  PROC DrawPart34()
    MoveL Offs(pOrigin,325.18,181.23,0.00),v40,z0,tPen\WObj:=wPaper;
    MoveL Offs(pOrigin,324.70,181.70,0.00),v40,z0,tPen\WObj:=wPaper;
    MoveL Offs(pOrigin,325.66,180.75,0.00),v40,z0,tPen\WObj:=wPaper;
    MoveL Offs(pOrigin,325.66,181.23,0.00),v40,z0,tPen\WObj:=wPaper;
    MoveL Offs(pOrigin,325.18,181.23,0.00),v40,z0,tPen\WObj:=wPaper;
    MoveL Offs(pOrigin,324.70,181.70,0.00),v40,fine,tPen\WObj:=wPaper;
    MoveL Offs(pOrigin,324.70,181.70,6.00),v60,z5,tPen\WObj:=wPaper;
    MoveL Offs(pOrigin,326.14,180.27,6.00),vTravel,z5,tPen\WObj:=wPaper;
    MoveL Offs(pOrigin,326.14,180.27,0.00),v60,z0,tPen\WObj:=wPaper;
    MoveL Offs(pOrigin,327.10,179.31,0.00),v40,z0,tPen\WObj:=wPaper;
    MoveL Offs(pOrigin,327.10,179.79,0.00),v40,z0,tPen\WObj:=wPaper;
    MoveL Offs(pOrigin,326.62,179.79,0.00),v40,z0,tPen\WObj:=wPaper;
    MoveL Offs(pOrigin,326.14,180.27,0.00),v40,z0,tPen\WObj:=wPaper;
    MoveL Offs(pOrigin,327.10,179.31,0.00),v40,z0,tPen\WObj:=wPaper;
    MoveL Offs(pOrigin,327.10,179.79,0.00),v40,z0,tPen\WObj:=wPaper;
    MoveL Offs(pOrigin,326.62,179.79,0.00),v40,z0,tPen\WObj:=wPaper;
    MoveL Offs(pOrigin,326.14,180.27,0.00),v40,fine,tPen\WObj:=wPaper;
    MoveL Offs(pOrigin,326.14,180.27,6.00),v60,z5,tPen\WObj:=wPaper;
    MoveL Offs(pOrigin,287.35,170.21,6.00),vTravel,z5,tPen\WObj:=wPaper;
    MoveL Offs(pOrigin,287.35,170.21,0.00),v60,z0,tPen\WObj:=wPaper;
    MoveL Offs(pOrigin,288.31,171.17,0.00),v40,z0,tPen\WObj:=wPaper;
    MoveL Offs(pOrigin,287.35,170.21,0.00),v40,fine,tPen\WObj:=wPaper;
    MoveL Offs(pOrigin,287.35,170.21,6.00),v60,z5,tPen\WObj:=wPaper;
    MoveL Offs(pOrigin,283.52,160.63,6.00),vTravel,z5,tPen\WObj:=wPaper;
    MoveL Offs(pOrigin,283.52,160.63,0.00),v60,z0,tPen\WObj:=wPaper;
    MoveL Offs(pOrigin,283.04,159.68,0.00),v40,z0,tPen\WObj:=wPaper;
    MoveL Offs(pOrigin,283.52,160.15,0.00),v40,z0,tPen\WObj:=wPaper;
    MoveL Offs(pOrigin,283.52,160.63,0.00),v40,z0,tPen\WObj:=wPaper;
    MoveL Offs(pOrigin,283.04,159.68,0.00),v40,z0,tPen\WObj:=wPaper;
    MoveL Offs(pOrigin,283.52,160.15,0.00),v40,z0,tPen\WObj:=wPaper;
    MoveL Offs(pOrigin,283.52,160.63,0.00),v40,fine,tPen\WObj:=wPaper;
    MoveL Offs(pOrigin,283.52,160.63,6.00),v60,z5,tPen\WObj:=wPaper;
    MoveL Offs(pOrigin,282.56,158.72,6.00),vTravel,z5,tPen\WObj:=wPaper;
    MoveL Offs(pOrigin,282.56,158.72,0.00),v60,z0,tPen\WObj:=wPaper;
    MoveL Offs(pOrigin,282.08,157.76,0.00),v40,z0,tPen\WObj:=wPaper;
    MoveL Offs(pOrigin,282.56,158.24,0.00),v40,z0,tPen\WObj:=wPaper;
    MoveL Offs(pOrigin,282.56,158.72,0.00),v40,z0,tPen\WObj:=wPaper;
    MoveL Offs(pOrigin,282.08,157.76,0.00),v40,z0,tPen\WObj:=wPaper;
    MoveL Offs(pOrigin,282.56,158.24,0.00),v40,z0,tPen\WObj:=wPaper;
    MoveL Offs(pOrigin,282.56,158.72,0.00),v40,fine,tPen\WObj:=wPaper;
    MoveL Offs(pOrigin,282.56,158.72,6.00),v60,z5,tPen\WObj:=wPaper;
    MoveL Offs(pOrigin,276.82,149.62,6.00),vTravel,z5,tPen\WObj:=wPaper;
    MoveL Offs(pOrigin,276.82,149.62,0.00),v60,z0,tPen\WObj:=wPaper;
    MoveL Offs(pOrigin,277.77,150.58,0.00),v40,z0,tPen\WObj:=wPaper;
    MoveL Offs(pOrigin,276.82,149.62,0.00),v40,fine,tPen\WObj:=wPaper;
    MoveL Offs(pOrigin,276.82,149.62,6.00),v60,z5,tPen\WObj:=wPaper;
    MoveL Offs(pOrigin,275.38,147.70,6.00),vTravel,z5,tPen\WObj:=wPaper;
    MoveL Offs(pOrigin,275.38,147.70,0.00),v60,z0,tPen\WObj:=wPaper;
    MoveL Offs(pOrigin,276.34,148.66,0.00),v40,z0,tPen\WObj:=wPaper;
    MoveL Offs(pOrigin,275.38,147.70,0.00),v40,fine,tPen\WObj:=wPaper;
    MoveL Offs(pOrigin,275.38,147.70,6.00),v60,z5,tPen\WObj:=wPaper;
    MoveL Offs(pOrigin,300.28,147.23,6.00),vTravel,z5,tPen\WObj:=wPaper;
    MoveL Offs(pOrigin,300.28,147.23,0.00),v60,z0,tPen\WObj:=wPaper;
    MoveL Offs(pOrigin,300.76,146.27,0.00),v40,z0,tPen\WObj:=wPaper;
    MoveL Offs(pOrigin,300.76,146.75,0.00),v40,z0,tPen\WObj:=wPaper;
    MoveL Offs(pOrigin,300.28,147.23,0.00),v40,z0,tPen\WObj:=wPaper;
    MoveL Offs(pOrigin,300.76,146.27,0.00),v40,z0,tPen\WObj:=wPaper;
    MoveL Offs(pOrigin,300.76,146.75,0.00),v40,z0,tPen\WObj:=wPaper;
    MoveL Offs(pOrigin,300.28,147.23,0.00),v40,fine,tPen\WObj:=wPaper;
    MoveL Offs(pOrigin,300.28,147.23,6.00),v60,z5,tPen\WObj:=wPaper;
    MoveL Offs(pOrigin,301.24,145.79,6.00),vTravel,z5,tPen\WObj:=wPaper;
    MoveL Offs(pOrigin,301.24,145.79,0.00),v60,z0,tPen\WObj:=wPaper;
    MoveL Offs(pOrigin,302.20,144.35,0.00),v40,z0,tPen\WObj:=wPaper;
    MoveL Offs(pOrigin,302.20,144.83,0.00),v40,z0,tPen\WObj:=wPaper;
    MoveL Offs(pOrigin,301.24,145.79,0.00),v40,z0,tPen\WObj:=wPaper;
    MoveL Offs(pOrigin,302.20,144.35,0.00),v40,z0,tPen\WObj:=wPaper;
    MoveL Offs(pOrigin,302.20,144.83,0.00),v40,z0,tPen\WObj:=wPaper;
    MoveL Offs(pOrigin,301.24,145.79,0.00),v40,fine,tPen\WObj:=wPaper;
    MoveL Offs(pOrigin,301.24,145.79,6.00),v60,z5,tPen\WObj:=wPaper;
    MoveL Offs(pOrigin,330.93,125.20,6.00),vTravel,z5,tPen\WObj:=wPaper;
    MoveL Offs(pOrigin,330.93,125.20,0.00),v60,z0,tPen\WObj:=wPaper;
    MoveL Offs(pOrigin,330.45,124.24,0.00),v40,z0,tPen\WObj:=wPaper;
    MoveL Offs(pOrigin,330.93,124.72,0.00),v40,z0,tPen\WObj:=wPaper;
    MoveL Offs(pOrigin,330.93,125.20,0.00),v40,z0,tPen\WObj:=wPaper;
    MoveL Offs(pOrigin,330.45,124.24,0.00),v40,z0,tPen\WObj:=wPaper;
    MoveL Offs(pOrigin,330.93,124.72,0.00),v40,z0,tPen\WObj:=wPaper;
    MoveL Offs(pOrigin,330.93,125.20,0.00),v40,fine,tPen\WObj:=wPaper;
    MoveL Offs(pOrigin,330.93,125.20,6.00),v60,z5,tPen\WObj:=wPaper;
    MoveL Offs(pOrigin,373.07,203.73,6.00),vTravel,z5,tPen\WObj:=wPaper;
    MoveL Offs(pOrigin,373.07,203.73,0.00),v60,z0,tPen\WObj:=wPaper;
    MoveL Offs(pOrigin,373.07,204.21,0.00),v40,z0,tPen\WObj:=wPaper;
    MoveL Offs(pOrigin,373.55,204.21,0.00),v40,z0,tPen\WObj:=wPaper;
    MoveL Offs(pOrigin,373.07,203.73,0.00),v40,z0,tPen\WObj:=wPaper;
    MoveL Offs(pOrigin,373.07,204.21,0.00),v40,z0,tPen\WObj:=wPaper;
    MoveL Offs(pOrigin,373.55,204.21,0.00),v40,z0,tPen\WObj:=wPaper;
    MoveL Offs(pOrigin,373.07,203.73,0.00),v40,fine,tPen\WObj:=wPaper;
    MoveL Offs(pOrigin,373.07,203.73,6.00),v60,z5,tPen\WObj:=wPaper;
    MoveL Offs(pOrigin,300.28,264.55,6.00),vTravel,z5,tPen\WObj:=wPaper;
    MoveL Offs(pOrigin,300.28,264.55,0.00),v60,z0,tPen\WObj:=wPaper;
    MoveL Offs(pOrigin,300.28,265.03,0.00),v40,z0,tPen\WObj:=wPaper;
    MoveL Offs(pOrigin,299.32,265.99,0.00),v40,z0,tPen\WObj:=wPaper;
    MoveL Offs(pOrigin,300.28,264.55,0.00),v40,z0,tPen\WObj:=wPaper;
    MoveL Offs(pOrigin,300.28,265.03,0.00),v40,z0,tPen\WObj:=wPaper;
    MoveL Offs(pOrigin,299.32,265.99,0.00),v40,z0,tPen\WObj:=wPaper;
    MoveL Offs(pOrigin,300.28,264.55,0.00),v40,fine,tPen\WObj:=wPaper;
    MoveL Offs(pOrigin,300.28,264.55,6.00),v60,z5,tPen\WObj:=wPaper;
    MoveL Offs(pOrigin,297.89,267.90,6.00),vTravel,z5,tPen\WObj:=wPaper;
    MoveL Offs(pOrigin,297.89,267.90,0.00),v60,z0,tPen\WObj:=wPaper;
    MoveL Offs(pOrigin,297.89,268.38,0.00),v40,z0,tPen\WObj:=wPaper;
    MoveL Offs(pOrigin,297.41,268.38,0.00),v40,z0,tPen\WObj:=wPaper;
    MoveL Offs(pOrigin,297.89,267.90,0.00),v40,z0,tPen\WObj:=wPaper;
    MoveL Offs(pOrigin,297.89,268.38,0.00),v40,z0,tPen\WObj:=wPaper;
    MoveL Offs(pOrigin,297.41,268.38,0.00),v40,z0,tPen\WObj:=wPaper;
    MoveL Offs(pOrigin,297.89,267.90,0.00),v40,fine,tPen\WObj:=wPaper;
    MoveL Offs(pOrigin,297.89,267.90,6.00),v60,z5,tPen\WObj:=wPaper;
    MoveL Offs(pOrigin,284.48,269.34,6.00),vTravel,z5,tPen\WObj:=wPaper;
    MoveL Offs(pOrigin,284.48,269.34,0.00),v60,z0,tPen\WObj:=wPaper;
    MoveL Offs(pOrigin,284.00,268.86,0.00),v40,z0,tPen\WObj:=wPaper;
    MoveL Offs(pOrigin,284.00,269.34,0.00),v40,z0,tPen\WObj:=wPaper;
    MoveL Offs(pOrigin,284.48,269.34,0.00),v40,z0,tPen\WObj:=wPaper;
    MoveL Offs(pOrigin,284.00,268.86,0.00),v40,z0,tPen\WObj:=wPaper;
    MoveL Offs(pOrigin,284.00,269.34,0.00),v40,z0,tPen\WObj:=wPaper;
    MoveL Offs(pOrigin,284.48,269.34,0.00),v40,fine,tPen\WObj:=wPaper;
    MoveL Offs(pOrigin,284.48,269.34,6.00),v60,z5,tPen\WObj:=wPaper;
    MoveL Offs(pOrigin,282.08,266.94,6.00),vTravel,z5,tPen\WObj:=wPaper;
    MoveL Offs(pOrigin,282.08,266.94,0.00),v60,z0,tPen\WObj:=wPaper;
    MoveL Offs(pOrigin,280.17,264.55,0.00),v40,z0,tPen\WObj:=wPaper;
    MoveL Offs(pOrigin,280.17,265.03,0.00),v40,z0,tPen\WObj:=wPaper;
    MoveL Offs(pOrigin,282.08,266.94,0.00),v40,z0,tPen\WObj:=wPaper;
    MoveL Offs(pOrigin,280.17,264.55,0.00),v40,z0,tPen\WObj:=wPaper;
  ENDPROC

  PROC DrawPart35()
    MoveL Offs(pOrigin,280.17,265.03,0.00),v40,z0,tPen\WObj:=wPaper;
    MoveL Offs(pOrigin,282.08,266.94,0.00),v40,fine,tPen\WObj:=wPaper;
    MoveL Offs(pOrigin,282.08,266.94,6.00),v60,z5,tPen\WObj:=wPaper;
    MoveL Offs(pOrigin,272.03,264.55,6.00),vTravel,z5,tPen\WObj:=wPaper;
    MoveL Offs(pOrigin,272.03,264.55,0.00),v60,z0,tPen\WObj:=wPaper;
    MoveL Offs(pOrigin,271.55,263.59,0.00),v40,z0,tPen\WObj:=wPaper;
    MoveL Offs(pOrigin,271.55,264.07,0.00),v40,z0,tPen\WObj:=wPaper;
    MoveL Offs(pOrigin,272.03,264.55,0.00),v40,z0,tPen\WObj:=wPaper;
    MoveL Offs(pOrigin,271.55,263.59,0.00),v40,z0,tPen\WObj:=wPaper;
    MoveL Offs(pOrigin,271.55,264.07,0.00),v40,z0,tPen\WObj:=wPaper;
    MoveL Offs(pOrigin,272.03,264.55,0.00),v40,fine,tPen\WObj:=wPaper;
    MoveL Offs(pOrigin,272.03,264.55,6.00),v60,z5,tPen\WObj:=wPaper;
    MoveL Offs(pOrigin,243.77,256.41,6.00),vTravel,z5,tPen\WObj:=wPaper;
    MoveL Offs(pOrigin,243.77,256.41,0.00),v60,z0,tPen\WObj:=wPaper;
    MoveL Offs(pOrigin,243.30,256.89,0.00),v40,z0,tPen\WObj:=wPaper;
    MoveL Offs(pOrigin,243.77,255.93,0.00),v40,z0,tPen\WObj:=wPaper;
    MoveL Offs(pOrigin,243.77,256.41,0.00),v40,z0,tPen\WObj:=wPaper;
    MoveL Offs(pOrigin,243.30,256.89,0.00),v40,z0,tPen\WObj:=wPaper;
    MoveL Offs(pOrigin,243.77,255.93,0.00),v40,z0,tPen\WObj:=wPaper;
    MoveL Offs(pOrigin,243.77,256.41,0.00),v40,fine,tPen\WObj:=wPaper;
    MoveL Offs(pOrigin,243.77,256.41,6.00),v60,z5,tPen\WObj:=wPaper;
    MoveL Offs(pOrigin,243.30,251.14,6.00),vTravel,z5,tPen\WObj:=wPaper;
    MoveL Offs(pOrigin,243.30,251.14,0.00),v60,z0,tPen\WObj:=wPaper;
    MoveL Offs(pOrigin,242.82,250.18,0.00),v40,z0,tPen\WObj:=wPaper;
    MoveL Offs(pOrigin,242.82,250.66,0.00),v40,z0,tPen\WObj:=wPaper;
    MoveL Offs(pOrigin,243.30,251.14,0.00),v40,z0,tPen\WObj:=wPaper;
    MoveL Offs(pOrigin,242.82,250.18,0.00),v40,z0,tPen\WObj:=wPaper;
    MoveL Offs(pOrigin,242.82,250.66,0.00),v40,z0,tPen\WObj:=wPaper;
    MoveL Offs(pOrigin,243.30,251.14,0.00),v40,fine,tPen\WObj:=wPaper;
    MoveL Offs(pOrigin,243.30,251.14,6.00),v60,z5,tPen\WObj:=wPaper;
    MoveL Offs(pOrigin,202.11,285.14,6.00),vTravel,z5,tPen\WObj:=wPaper;
    MoveL Offs(pOrigin,202.11,285.14,0.00),v60,z0,tPen\WObj:=wPaper;
    MoveL Offs(pOrigin,201.15,284.66,0.00),v40,z0,tPen\WObj:=wPaper;
    MoveL Offs(pOrigin,201.63,284.66,0.00),v40,z0,tPen\WObj:=wPaper;
    MoveL Offs(pOrigin,202.11,285.14,0.00),v40,z0,tPen\WObj:=wPaper;
    MoveL Offs(pOrigin,201.15,284.66,0.00),v40,z0,tPen\WObj:=wPaper;
    MoveL Offs(pOrigin,201.63,284.66,0.00),v40,z0,tPen\WObj:=wPaper;
    MoveL Offs(pOrigin,202.11,285.14,0.00),v40,fine,tPen\WObj:=wPaper;
    MoveL Offs(pOrigin,202.11,285.14,6.00),v60,z5,tPen\WObj:=wPaper;
    MoveL Offs(pOrigin,197.32,282.75,6.00),vTravel,z5,tPen\WObj:=wPaper;
    MoveL Offs(pOrigin,197.32,282.75,0.00),v60,z0,tPen\WObj:=wPaper;
    MoveL Offs(pOrigin,195.89,281.79,0.00),v40,z0,tPen\WObj:=wPaper;
    MoveL Offs(pOrigin,196.37,281.79,0.00),v40,z0,tPen\WObj:=wPaper;
    MoveL Offs(pOrigin,197.32,282.75,0.00),v40,z0,tPen\WObj:=wPaper;
    MoveL Offs(pOrigin,195.89,281.79,0.00),v40,z0,tPen\WObj:=wPaper;
    MoveL Offs(pOrigin,196.37,281.79,0.00),v40,z0,tPen\WObj:=wPaper;
    MoveL Offs(pOrigin,197.32,282.75,0.00),v40,fine,tPen\WObj:=wPaper;
    MoveL Offs(pOrigin,197.32,282.75,6.00),v60,z5,tPen\WObj:=wPaper;
    MoveL Offs(pOrigin,193.97,280.83,6.00),vTravel,z5,tPen\WObj:=wPaper;
    MoveL Offs(pOrigin,193.97,280.83,0.00),v60,z0,tPen\WObj:=wPaper;
    MoveL Offs(pOrigin,193.01,280.35,0.00),v40,z0,tPen\WObj:=wPaper;
    MoveL Offs(pOrigin,193.49,280.35,0.00),v40,z0,tPen\WObj:=wPaper;
    MoveL Offs(pOrigin,193.97,280.83,0.00),v40,z0,tPen\WObj:=wPaper;
    MoveL Offs(pOrigin,193.01,280.35,0.00),v40,z0,tPen\WObj:=wPaper;
    MoveL Offs(pOrigin,193.49,280.35,0.00),v40,z0,tPen\WObj:=wPaper;
    MoveL Offs(pOrigin,193.97,280.83,0.00),v40,fine,tPen\WObj:=wPaper;
    MoveL Offs(pOrigin,193.97,280.83,6.00),v60,z5,tPen\WObj:=wPaper;
    MoveL Offs(pOrigin,186.31,276.04,6.00),vTravel,z5,tPen\WObj:=wPaper;
    MoveL Offs(pOrigin,186.31,276.04,0.00),v60,z0,tPen\WObj:=wPaper;
    MoveL Offs(pOrigin,184.39,274.61,0.00),v40,z0,tPen\WObj:=wPaper;
    MoveL Offs(pOrigin,184.87,274.61,0.00),v40,z0,tPen\WObj:=wPaper;
    MoveL Offs(pOrigin,186.31,276.04,0.00),v40,z0,tPen\WObj:=wPaper;
    MoveL Offs(pOrigin,184.39,274.61,0.00),v40,z0,tPen\WObj:=wPaper;
    MoveL Offs(pOrigin,184.87,274.61,0.00),v40,z0,tPen\WObj:=wPaper;
    MoveL Offs(pOrigin,186.31,276.04,0.00),v40,fine,tPen\WObj:=wPaper;
    MoveL Offs(pOrigin,186.31,276.04,6.00),v60,z5,tPen\WObj:=wPaper;
    MoveL Offs(pOrigin,181.04,272.21,6.00),vTravel,z5,tPen\WObj:=wPaper;
    MoveL Offs(pOrigin,181.04,272.21,0.00),v60,z0,tPen\WObj:=wPaper;
    MoveL Offs(pOrigin,179.13,270.77,0.00),v40,z0,tPen\WObj:=wPaper;
    MoveL Offs(pOrigin,179.61,270.77,0.00),v40,z0,tPen\WObj:=wPaper;
    MoveL Offs(pOrigin,181.04,272.21,0.00),v40,z0,tPen\WObj:=wPaper;
    MoveL Offs(pOrigin,179.13,270.77,0.00),v40,z0,tPen\WObj:=wPaper;
    MoveL Offs(pOrigin,179.61,270.77,0.00),v40,z0,tPen\WObj:=wPaper;
    MoveL Offs(pOrigin,181.04,272.21,0.00),v40,fine,tPen\WObj:=wPaper;
    MoveL Offs(pOrigin,181.04,272.21,6.00),v60,z5,tPen\WObj:=wPaper;
    MoveL Offs(pOrigin,177.69,269.34,6.00),vTravel,z5,tPen\WObj:=wPaper;
    MoveL Offs(pOrigin,177.69,269.34,0.00),v60,z0,tPen\WObj:=wPaper;
    MoveL Offs(pOrigin,178.65,270.30,0.00),v40,z0,tPen\WObj:=wPaper;
    MoveL Offs(pOrigin,177.69,269.34,0.00),v40,fine,tPen\WObj:=wPaper;
    MoveL Offs(pOrigin,177.69,269.34,6.00),v60,z5,tPen\WObj:=wPaper;
    MoveL Offs(pOrigin,171.94,274.13,6.00),vTravel,z5,tPen\WObj:=wPaper;
    MoveL Offs(pOrigin,171.94,274.13,0.00),v60,z0,tPen\WObj:=wPaper;
    MoveL Offs(pOrigin,173.86,276.04,0.00),v40,z0,tPen\WObj:=wPaper;
    MoveL Offs(pOrigin,171.46,273.65,0.00),v40,z0,tPen\WObj:=wPaper;
    MoveL Offs(pOrigin,171.46,274.13,0.00),v40,z0,tPen\WObj:=wPaper;
    MoveL Offs(pOrigin,171.94,274.13,0.00),v40,z0,tPen\WObj:=wPaper;
    MoveL Offs(pOrigin,173.86,276.04,0.00),v40,z0,tPen\WObj:=wPaper;
    MoveL Offs(pOrigin,171.46,273.65,0.00),v40,z0,tPen\WObj:=wPaper;
    MoveL Offs(pOrigin,171.46,274.13,0.00),v40,z0,tPen\WObj:=wPaper;
    MoveL Offs(pOrigin,171.94,274.13,0.00),v40,fine,tPen\WObj:=wPaper;
    MoveL Offs(pOrigin,171.94,274.13,6.00),v60,z5,tPen\WObj:=wPaper;
    MoveL Offs(pOrigin,170.51,273.17,6.00),vTravel,z5,tPen\WObj:=wPaper;
    MoveL Offs(pOrigin,170.51,273.17,0.00),v60,z0,tPen\WObj:=wPaper;
    MoveL Offs(pOrigin,166.20,268.86,0.00),v40,z0,tPen\WObj:=wPaper;
    MoveL Offs(pOrigin,166.20,269.34,0.00),v40,z0,tPen\WObj:=wPaper;
    MoveL Offs(pOrigin,166.68,269.34,0.00),v40,z0,tPen\WObj:=wPaper;
    MoveL Offs(pOrigin,170.51,273.17,0.00),v40,z0,tPen\WObj:=wPaper;
    MoveL Offs(pOrigin,166.20,268.86,0.00),v40,z0,tPen\WObj:=wPaper;
    MoveL Offs(pOrigin,166.20,269.34,0.00),v40,z0,tPen\WObj:=wPaper;
    MoveL Offs(pOrigin,166.68,269.34,0.00),v40,z0,tPen\WObj:=wPaper;
    MoveL Offs(pOrigin,170.51,273.17,0.00),v40,fine,tPen\WObj:=wPaper;
    MoveL Offs(pOrigin,170.51,273.17,6.00),v60,z5,tPen\WObj:=wPaper;
    MoveL Offs(pOrigin,174.34,276.52,6.00),vTravel,z5,tPen\WObj:=wPaper;
    MoveL Offs(pOrigin,174.34,276.52,0.00),v60,z0,tPen\WObj:=wPaper;
    MoveL Offs(pOrigin,174.34,277.00,0.00),v40,z0,tPen\WObj:=wPaper;
    MoveL Offs(pOrigin,174.82,277.00,0.00),v40,z0,tPen\WObj:=wPaper;
    MoveL Offs(pOrigin,177.21,279.39,0.00),v40,z0,tPen\WObj:=wPaper;
    MoveL Offs(pOrigin,174.34,276.52,0.00),v40,z0,tPen\WObj:=wPaper;
    MoveL Offs(pOrigin,174.34,277.00,0.00),v40,z0,tPen\WObj:=wPaper;
    MoveL Offs(pOrigin,174.82,277.00,0.00),v40,z0,tPen\WObj:=wPaper;
    MoveL Offs(pOrigin,177.21,279.39,0.00),v40,z0,tPen\WObj:=wPaper;
    MoveL Offs(pOrigin,174.34,276.52,0.00),v40,fine,tPen\WObj:=wPaper;
    MoveL Offs(pOrigin,174.34,276.52,6.00),v60,z5,tPen\WObj:=wPaper;
    MoveL Offs(pOrigin,178.17,279.87,6.00),vTravel,z5,tPen\WObj:=wPaper;
    MoveL Offs(pOrigin,178.17,279.87,0.00),v60,z0,tPen\WObj:=wPaper;
    MoveL Offs(pOrigin,178.17,280.35,0.00),v40,z0,tPen\WObj:=wPaper;
    MoveL Offs(pOrigin,178.65,280.35,0.00),v40,z0,tPen\WObj:=wPaper;
    MoveL Offs(pOrigin,179.13,280.83,0.00),v40,z0,tPen\WObj:=wPaper;
    MoveL Offs(pOrigin,178.17,279.87,0.00),v40,z0,tPen\WObj:=wPaper;
    MoveL Offs(pOrigin,178.17,280.35,0.00),v40,z0,tPen\WObj:=wPaper;
  ENDPROC

  PROC DrawPart36()
    MoveL Offs(pOrigin,178.65,280.35,0.00),v40,z0,tPen\WObj:=wPaper;
    MoveL Offs(pOrigin,179.13,280.83,0.00),v40,z0,tPen\WObj:=wPaper;
    MoveL Offs(pOrigin,178.17,279.87,0.00),v40,fine,tPen\WObj:=wPaper;
    MoveL Offs(pOrigin,178.17,279.87,6.00),v60,z5,tPen\WObj:=wPaper;
    MoveL Offs(pOrigin,181.04,282.27,6.00),vTravel,z5,tPen\WObj:=wPaper;
    MoveL Offs(pOrigin,181.04,282.27,0.00),v60,z0,tPen\WObj:=wPaper;
    MoveL Offs(pOrigin,181.04,282.75,0.00),v40,z0,tPen\WObj:=wPaper;
    MoveL Offs(pOrigin,181.52,282.75,0.00),v40,z0,tPen\WObj:=wPaper;
    MoveL Offs(pOrigin,181.04,282.27,0.00),v40,z0,tPen\WObj:=wPaper;
    MoveL Offs(pOrigin,181.04,282.75,0.00),v40,z0,tPen\WObj:=wPaper;
    MoveL Offs(pOrigin,181.52,282.75,0.00),v40,z0,tPen\WObj:=wPaper;
    MoveL Offs(pOrigin,181.04,282.27,0.00),v40,fine,tPen\WObj:=wPaper;
    MoveL Offs(pOrigin,181.04,282.27,6.00),v60,z5,tPen\WObj:=wPaper;
    MoveL Offs(pOrigin,183.92,284.18,6.00),vTravel,z5,tPen\WObj:=wPaper;
    MoveL Offs(pOrigin,183.92,284.18,0.00),v60,z0,tPen\WObj:=wPaper;
    MoveL Offs(pOrigin,183.92,284.66,0.00),v40,z0,tPen\WObj:=wPaper;
    MoveL Offs(pOrigin,184.39,284.66,0.00),v40,z0,tPen\WObj:=wPaper;
    MoveL Offs(pOrigin,183.92,284.18,0.00),v40,z0,tPen\WObj:=wPaper;
    MoveL Offs(pOrigin,183.92,284.66,0.00),v40,z0,tPen\WObj:=wPaper;
    MoveL Offs(pOrigin,184.39,284.66,0.00),v40,z0,tPen\WObj:=wPaper;
    MoveL Offs(pOrigin,183.92,284.18,0.00),v40,fine,tPen\WObj:=wPaper;
    MoveL Offs(pOrigin,183.92,284.18,6.00),v60,z5,tPen\WObj:=wPaper;
    MoveL Offs(pOrigin,185.35,285.14,6.00),vTravel,z5,tPen\WObj:=wPaper;
    MoveL Offs(pOrigin,185.35,285.14,0.00),v60,z0,tPen\WObj:=wPaper;
    MoveL Offs(pOrigin,185.35,285.62,0.00),v40,z0,tPen\WObj:=wPaper;
    MoveL Offs(pOrigin,185.83,285.62,0.00),v40,z0,tPen\WObj:=wPaper;
    MoveL Offs(pOrigin,186.31,286.10,0.00),v40,z0,tPen\WObj:=wPaper;
    MoveL Offs(pOrigin,185.35,285.14,0.00),v40,z0,tPen\WObj:=wPaper;
    MoveL Offs(pOrigin,185.35,285.62,0.00),v40,z0,tPen\WObj:=wPaper;
    MoveL Offs(pOrigin,185.83,285.62,0.00),v40,z0,tPen\WObj:=wPaper;
    MoveL Offs(pOrigin,186.31,286.10,0.00),v40,z0,tPen\WObj:=wPaper;
    MoveL Offs(pOrigin,185.35,285.14,0.00),v40,fine,tPen\WObj:=wPaper;
    MoveL Offs(pOrigin,185.35,285.14,6.00),v60,z5,tPen\WObj:=wPaper;
    MoveL Offs(pOrigin,180.08,294.24,6.00),vTravel,z5,tPen\WObj:=wPaper;
    MoveL Offs(pOrigin,180.08,294.24,0.00),v60,z0,tPen\WObj:=wPaper;
    MoveL Offs(pOrigin,180.08,294.72,0.00),v40,z0,tPen\WObj:=wPaper;
    MoveL Offs(pOrigin,180.56,294.72,0.00),v40,z0,tPen\WObj:=wPaper;
    MoveL Offs(pOrigin,180.08,294.24,0.00),v40,z0,tPen\WObj:=wPaper;
    MoveL Offs(pOrigin,180.08,294.72,0.00),v40,z0,tPen\WObj:=wPaper;
    MoveL Offs(pOrigin,180.56,294.72,0.00),v40,z0,tPen\WObj:=wPaper;
    MoveL Offs(pOrigin,180.08,294.24,0.00),v40,fine,tPen\WObj:=wPaper;
    MoveL Offs(pOrigin,180.08,294.24,6.00),v60,z5,tPen\WObj:=wPaper;
    MoveL Offs(pOrigin,175.30,290.89,6.00),vTravel,z5,tPen\WObj:=wPaper;
    MoveL Offs(pOrigin,175.30,290.89,0.00),v60,z0,tPen\WObj:=wPaper;
    MoveL Offs(pOrigin,174.34,289.93,0.00),v40,z0,tPen\WObj:=wPaper;
    MoveL Offs(pOrigin,174.34,290.41,0.00),v40,z0,tPen\WObj:=wPaper;
    MoveL Offs(pOrigin,174.82,290.41,0.00),v40,z0,tPen\WObj:=wPaper;
    MoveL Offs(pOrigin,175.30,290.89,0.00),v40,z0,tPen\WObj:=wPaper;
    MoveL Offs(pOrigin,174.34,289.93,0.00),v40,z0,tPen\WObj:=wPaper;
    MoveL Offs(pOrigin,174.34,290.41,0.00),v40,z0,tPen\WObj:=wPaper;
    MoveL Offs(pOrigin,174.82,290.41,0.00),v40,z0,tPen\WObj:=wPaper;
    MoveL Offs(pOrigin,175.30,290.89,0.00),v40,fine,tPen\WObj:=wPaper;
    MoveL Offs(pOrigin,175.30,290.89,6.00),v60,z5,tPen\WObj:=wPaper;
    MoveL Offs(pOrigin,173.38,289.45,6.00),vTravel,z5,tPen\WObj:=wPaper;
    MoveL Offs(pOrigin,173.38,289.45,0.00),v60,z0,tPen\WObj:=wPaper;
    MoveL Offs(pOrigin,172.42,288.49,0.00),v40,z0,tPen\WObj:=wPaper;
    MoveL Offs(pOrigin,172.42,288.97,0.00),v40,z0,tPen\WObj:=wPaper;
    MoveL Offs(pOrigin,172.90,288.97,0.00),v40,z0,tPen\WObj:=wPaper;
    MoveL Offs(pOrigin,173.38,289.45,0.00),v40,z0,tPen\WObj:=wPaper;
    MoveL Offs(pOrigin,172.42,288.49,0.00),v40,z0,tPen\WObj:=wPaper;
    MoveL Offs(pOrigin,172.42,288.97,0.00),v40,z0,tPen\WObj:=wPaper;
    MoveL Offs(pOrigin,172.90,288.97,0.00),v40,z0,tPen\WObj:=wPaper;
    MoveL Offs(pOrigin,173.38,289.45,0.00),v40,fine,tPen\WObj:=wPaper;
    MoveL Offs(pOrigin,173.38,289.45,6.00),v60,z5,tPen\WObj:=wPaper;
    MoveL Offs(pOrigin,171.46,288.01,6.00),vTravel,z5,tPen\WObj:=wPaper;
    MoveL Offs(pOrigin,171.46,288.01,0.00),v60,z0,tPen\WObj:=wPaper;
    MoveL Offs(pOrigin,169.55,286.10,0.00),v40,z0,tPen\WObj:=wPaper;
    MoveL Offs(pOrigin,169.55,286.58,0.00),v40,z0,tPen\WObj:=wPaper;
    MoveL Offs(pOrigin,170.03,286.58,0.00),v40,z0,tPen\WObj:=wPaper;
    MoveL Offs(pOrigin,171.46,288.01,0.00),v40,z0,tPen\WObj:=wPaper;
    MoveL Offs(pOrigin,169.55,286.10,0.00),v40,z0,tPen\WObj:=wPaper;
    MoveL Offs(pOrigin,169.55,286.58,0.00),v40,z0,tPen\WObj:=wPaper;
    MoveL Offs(pOrigin,170.03,286.58,0.00),v40,z0,tPen\WObj:=wPaper;
    MoveL Offs(pOrigin,171.46,288.01,0.00),v40,fine,tPen\WObj:=wPaper;
    MoveL Offs(pOrigin,171.46,288.01,6.00),v60,z5,tPen\WObj:=wPaper;
    MoveL Offs(pOrigin,168.59,285.62,6.00),vTravel,z5,tPen\WObj:=wPaper;
    MoveL Offs(pOrigin,168.59,285.62,0.00),v60,z0,tPen\WObj:=wPaper;
    MoveL Offs(pOrigin,166.20,283.23,0.00),v40,z0,tPen\WObj:=wPaper;
    MoveL Offs(pOrigin,166.20,283.70,0.00),v40,z0,tPen\WObj:=wPaper;
    MoveL Offs(pOrigin,166.68,283.70,0.00),v40,z0,tPen\WObj:=wPaper;
    MoveL Offs(pOrigin,168.59,285.62,0.00),v40,z0,tPen\WObj:=wPaper;
    MoveL Offs(pOrigin,166.20,283.23,0.00),v40,z0,tPen\WObj:=wPaper;
    MoveL Offs(pOrigin,166.20,283.70,0.00),v40,z0,tPen\WObj:=wPaper;
    MoveL Offs(pOrigin,166.68,283.70,0.00),v40,z0,tPen\WObj:=wPaper;
    MoveL Offs(pOrigin,168.59,285.62,0.00),v40,fine,tPen\WObj:=wPaper;
    MoveL Offs(pOrigin,168.59,285.62,6.00),v60,z5,tPen\WObj:=wPaper;
    MoveL Offs(pOrigin,165.72,282.75,6.00),vTravel,z5,tPen\WObj:=wPaper;
    MoveL Offs(pOrigin,165.72,282.75,0.00),v60,z0,tPen\WObj:=wPaper;
    MoveL Offs(pOrigin,164.76,281.79,0.00),v40,z0,tPen\WObj:=wPaper;
    MoveL Offs(pOrigin,164.76,282.27,0.00),v40,z0,tPen\WObj:=wPaper;
    MoveL Offs(pOrigin,165.24,282.27,0.00),v40,z0,tPen\WObj:=wPaper;
    MoveL Offs(pOrigin,165.72,282.75,0.00),v40,z0,tPen\WObj:=wPaper;
    MoveL Offs(pOrigin,164.76,281.79,0.00),v40,z0,tPen\WObj:=wPaper;
    MoveL Offs(pOrigin,164.76,282.27,0.00),v40,z0,tPen\WObj:=wPaper;
    MoveL Offs(pOrigin,165.24,282.27,0.00),v40,z0,tPen\WObj:=wPaper;
    MoveL Offs(pOrigin,165.72,282.75,0.00),v40,fine,tPen\WObj:=wPaper;
    MoveL Offs(pOrigin,165.72,282.75,6.00),v60,z5,tPen\WObj:=wPaper;
    MoveL Offs(pOrigin,163.80,281.31,6.00),vTravel,z5,tPen\WObj:=wPaper;
    MoveL Offs(pOrigin,163.80,281.31,0.00),v60,z0,tPen\WObj:=wPaper;
    MoveL Offs(pOrigin,163.32,280.83,0.00),v40,z0,tPen\WObj:=wPaper;
    MoveL Offs(pOrigin,163.32,281.31,0.00),v40,z0,tPen\WObj:=wPaper;
    MoveL Offs(pOrigin,163.80,281.31,0.00),v40,z0,tPen\WObj:=wPaper;
    MoveL Offs(pOrigin,163.32,280.83,0.00),v40,z0,tPen\WObj:=wPaper;
    MoveL Offs(pOrigin,163.32,281.31,0.00),v40,z0,tPen\WObj:=wPaper;
    MoveL Offs(pOrigin,163.80,281.31,0.00),v40,fine,tPen\WObj:=wPaper;
    MoveL Offs(pOrigin,163.80,281.31,6.00),v60,z5,tPen\WObj:=wPaper;
    MoveL Offs(pOrigin,162.37,279.87,6.00),vTravel,z5,tPen\WObj:=wPaper;
    MoveL Offs(pOrigin,162.37,279.87,0.00),v60,z0,tPen\WObj:=wPaper;
    MoveL Offs(pOrigin,158.54,276.04,0.00),v40,z0,tPen\WObj:=wPaper;
    MoveL Offs(pOrigin,158.54,276.52,0.00),v40,z0,tPen\WObj:=wPaper;
    MoveL Offs(pOrigin,159.01,276.52,0.00),v40,z0,tPen\WObj:=wPaper;
    MoveL Offs(pOrigin,162.37,279.87,0.00),v40,z0,tPen\WObj:=wPaper;
    MoveL Offs(pOrigin,158.54,276.04,0.00),v40,z0,tPen\WObj:=wPaper;
    MoveL Offs(pOrigin,158.54,276.52,0.00),v40,z0,tPen\WObj:=wPaper;
    MoveL Offs(pOrigin,159.01,276.52,0.00),v40,z0,tPen\WObj:=wPaper;
    MoveL Offs(pOrigin,162.37,279.87,0.00),v40,fine,tPen\WObj:=wPaper;
    MoveL Offs(pOrigin,162.37,279.87,6.00),v60,z5,tPen\WObj:=wPaper;
    MoveL Offs(pOrigin,158.06,275.08,6.00),vTravel,z5,tPen\WObj:=wPaper;
    MoveL Offs(pOrigin,158.06,275.08,0.00),v60,z0,tPen\WObj:=wPaper;
    MoveL Offs(pOrigin,156.62,273.65,0.00),v40,z0,tPen\WObj:=wPaper;
  ENDPROC

  PROC DrawPart37()
    MoveL Offs(pOrigin,156.62,274.13,0.00),v40,z0,tPen\WObj:=wPaper;
    MoveL Offs(pOrigin,157.10,274.13,0.00),v40,z0,tPen\WObj:=wPaper;
    MoveL Offs(pOrigin,158.06,275.08,0.00),v40,z0,tPen\WObj:=wPaper;
    MoveL Offs(pOrigin,156.62,273.65,0.00),v40,z0,tPen\WObj:=wPaper;
    MoveL Offs(pOrigin,156.62,274.13,0.00),v40,z0,tPen\WObj:=wPaper;
    MoveL Offs(pOrigin,157.10,274.13,0.00),v40,z0,tPen\WObj:=wPaper;
    MoveL Offs(pOrigin,158.06,275.08,0.00),v40,fine,tPen\WObj:=wPaper;
    MoveL Offs(pOrigin,158.06,275.08,6.00),v60,z5,tPen\WObj:=wPaper;
    MoveL Offs(pOrigin,155.18,271.73,6.00),vTravel,z5,tPen\WObj:=wPaper;
    MoveL Offs(pOrigin,155.18,271.73,0.00),v60,z0,tPen\WObj:=wPaper;
    MoveL Offs(pOrigin,153.75,270.30,0.00),v40,z0,tPen\WObj:=wPaper;
    MoveL Offs(pOrigin,153.75,270.77,0.00),v40,z0,tPen\WObj:=wPaper;
    MoveL Offs(pOrigin,154.23,270.77,0.00),v40,z0,tPen\WObj:=wPaper;
    MoveL Offs(pOrigin,155.18,271.73,0.00),v40,z0,tPen\WObj:=wPaper;
    MoveL Offs(pOrigin,153.75,270.30,0.00),v40,z0,tPen\WObj:=wPaper;
    MoveL Offs(pOrigin,153.75,270.77,0.00),v40,z0,tPen\WObj:=wPaper;
    MoveL Offs(pOrigin,154.23,270.77,0.00),v40,z0,tPen\WObj:=wPaper;
    MoveL Offs(pOrigin,155.18,271.73,0.00),v40,fine,tPen\WObj:=wPaper;
    MoveL Offs(pOrigin,155.18,271.73,6.00),v60,z5,tPen\WObj:=wPaper;
    MoveL Offs(pOrigin,152.79,268.86,6.00),vTravel,z5,tPen\WObj:=wPaper;
    MoveL Offs(pOrigin,152.79,268.86,0.00),v60,z0,tPen\WObj:=wPaper;
    MoveL Offs(pOrigin,151.35,266.94,0.00),v40,z0,tPen\WObj:=wPaper;
    MoveL Offs(pOrigin,151.35,267.42,0.00),v40,z0,tPen\WObj:=wPaper;
    MoveL Offs(pOrigin,152.79,268.86,0.00),v40,z0,tPen\WObj:=wPaper;
    MoveL Offs(pOrigin,151.35,266.94,0.00),v40,z0,tPen\WObj:=wPaper;
    MoveL Offs(pOrigin,151.35,267.42,0.00),v40,z0,tPen\WObj:=wPaper;
    MoveL Offs(pOrigin,152.79,268.86,0.00),v40,fine,tPen\WObj:=wPaper;
    MoveL Offs(pOrigin,152.79,268.86,6.00),v60,z5,tPen\WObj:=wPaper;
    MoveL Offs(pOrigin,149.92,265.03,6.00),vTravel,z5,tPen\WObj:=wPaper;
    MoveL Offs(pOrigin,149.92,265.03,0.00),v60,z0,tPen\WObj:=wPaper;
    MoveL Offs(pOrigin,149.44,264.55,0.00),v40,z0,tPen\WObj:=wPaper;
    MoveL Offs(pOrigin,149.44,265.03,0.00),v40,z0,tPen\WObj:=wPaper;
    MoveL Offs(pOrigin,149.92,265.03,0.00),v40,z0,tPen\WObj:=wPaper;
    MoveL Offs(pOrigin,149.44,264.55,0.00),v40,z0,tPen\WObj:=wPaper;
    MoveL Offs(pOrigin,149.44,265.03,0.00),v40,z0,tPen\WObj:=wPaper;
    MoveL Offs(pOrigin,149.92,265.03,0.00),v40,fine,tPen\WObj:=wPaper;
    MoveL Offs(pOrigin,149.92,265.03,6.00),v60,z5,tPen\WObj:=wPaper;
    MoveL Offs(pOrigin,147.52,261.68,6.00),vTravel,z5,tPen\WObj:=wPaper;
    MoveL Offs(pOrigin,147.52,261.68,0.00),v60,z0,tPen\WObj:=wPaper;
    MoveL Offs(pOrigin,146.56,260.72,0.00),v40,z0,tPen\WObj:=wPaper;
    MoveL Offs(pOrigin,146.56,261.20,0.00),v40,z0,tPen\WObj:=wPaper;
    MoveL Offs(pOrigin,147.04,261.20,0.00),v40,z0,tPen\WObj:=wPaper;
    MoveL Offs(pOrigin,147.52,261.68,0.00),v40,z0,tPen\WObj:=wPaper;
    MoveL Offs(pOrigin,146.56,260.72,0.00),v40,z0,tPen\WObj:=wPaper;
    MoveL Offs(pOrigin,146.56,261.20,0.00),v40,z0,tPen\WObj:=wPaper;
    MoveL Offs(pOrigin,147.04,261.20,0.00),v40,z0,tPen\WObj:=wPaper;
    MoveL Offs(pOrigin,147.52,261.68,0.00),v40,fine,tPen\WObj:=wPaper;
    MoveL Offs(pOrigin,147.52,261.68,6.00),v60,z5,tPen\WObj:=wPaper;
    MoveL Offs(pOrigin,145.61,258.80,6.00),vTravel,z5,tPen\WObj:=wPaper;
    MoveL Offs(pOrigin,145.61,258.80,0.00),v60,z0,tPen\WObj:=wPaper;
    MoveL Offs(pOrigin,144.65,257.37,0.00),v40,z0,tPen\WObj:=wPaper;
    MoveL Offs(pOrigin,144.65,257.85,0.00),v40,z0,tPen\WObj:=wPaper;
    MoveL Offs(pOrigin,145.61,258.80,0.00),v40,z0,tPen\WObj:=wPaper;
    MoveL Offs(pOrigin,144.65,257.37,0.00),v40,z0,tPen\WObj:=wPaper;
    MoveL Offs(pOrigin,144.65,257.85,0.00),v40,z0,tPen\WObj:=wPaper;
    MoveL Offs(pOrigin,145.61,258.80,0.00),v40,fine,tPen\WObj:=wPaper;
    MoveL Offs(pOrigin,145.61,258.80,6.00),v60,z5,tPen\WObj:=wPaper;
    MoveL Offs(pOrigin,142.73,254.01,6.00),vTravel,z5,tPen\WObj:=wPaper;
    MoveL Offs(pOrigin,142.73,254.01,0.00),v60,z0,tPen\WObj:=wPaper;
    MoveL Offs(pOrigin,142.25,253.54,0.00),v40,z0,tPen\WObj:=wPaper;
    MoveL Offs(pOrigin,142.25,254.01,0.00),v40,z0,tPen\WObj:=wPaper;
    MoveL Offs(pOrigin,142.73,254.01,0.00),v40,z0,tPen\WObj:=wPaper;
    MoveL Offs(pOrigin,142.25,253.54,0.00),v40,z0,tPen\WObj:=wPaper;
    MoveL Offs(pOrigin,142.25,254.01,0.00),v40,z0,tPen\WObj:=wPaper;
    MoveL Offs(pOrigin,142.73,254.01,0.00),v40,fine,tPen\WObj:=wPaper;
    MoveL Offs(pOrigin,142.73,254.01,6.00),v60,z5,tPen\WObj:=wPaper;
    MoveL Offs(pOrigin,141.30,251.62,6.00),vTravel,z5,tPen\WObj:=wPaper;
    MoveL Offs(pOrigin,141.30,251.62,0.00),v60,z0,tPen\WObj:=wPaper;
    MoveL Offs(pOrigin,140.82,251.14,0.00),v40,z0,tPen\WObj:=wPaper;
    MoveL Offs(pOrigin,140.82,251.62,0.00),v40,z0,tPen\WObj:=wPaper;
    MoveL Offs(pOrigin,141.30,251.62,0.00),v40,z0,tPen\WObj:=wPaper;
    MoveL Offs(pOrigin,140.82,251.14,0.00),v40,z0,tPen\WObj:=wPaper;
    MoveL Offs(pOrigin,140.82,251.62,0.00),v40,z0,tPen\WObj:=wPaper;
    MoveL Offs(pOrigin,141.30,251.62,0.00),v40,fine,tPen\WObj:=wPaper;
    MoveL Offs(pOrigin,141.30,251.62,6.00),v60,z5,tPen\WObj:=wPaper;
    MoveL Offs(pOrigin,140.34,249.70,6.00),vTravel,z5,tPen\WObj:=wPaper;
    MoveL Offs(pOrigin,140.34,249.70,0.00),v60,z0,tPen\WObj:=wPaper;
    MoveL Offs(pOrigin,139.86,249.23,0.00),v40,z0,tPen\WObj:=wPaper;
    MoveL Offs(pOrigin,139.86,249.70,0.00),v40,z0,tPen\WObj:=wPaper;
    MoveL Offs(pOrigin,140.34,249.70,0.00),v40,z0,tPen\WObj:=wPaper;
    MoveL Offs(pOrigin,139.86,249.23,0.00),v40,z0,tPen\WObj:=wPaper;
    MoveL Offs(pOrigin,139.86,249.70,0.00),v40,z0,tPen\WObj:=wPaper;
    MoveL Offs(pOrigin,140.34,249.70,0.00),v40,fine,tPen\WObj:=wPaper;
    MoveL Offs(pOrigin,140.34,249.70,6.00),v60,z5,tPen\WObj:=wPaper;
    MoveL Offs(pOrigin,133.15,253.06,6.00),vTravel,z5,tPen\WObj:=wPaper;
    MoveL Offs(pOrigin,133.15,253.06,0.00),v60,z0,tPen\WObj:=wPaper;
    MoveL Offs(pOrigin,133.15,253.54,0.00),v40,z0,tPen\WObj:=wPaper;
    MoveL Offs(pOrigin,132.68,252.58,0.00),v40,z0,tPen\WObj:=wPaper;
    MoveL Offs(pOrigin,133.15,253.06,0.00),v40,z0,tPen\WObj:=wPaper;
    MoveL Offs(pOrigin,133.15,253.54,0.00),v40,z0,tPen\WObj:=wPaper;
    MoveL Offs(pOrigin,132.68,252.58,0.00),v40,z0,tPen\WObj:=wPaper;
    MoveL Offs(pOrigin,133.15,253.06,0.00),v40,fine,tPen\WObj:=wPaper;
    MoveL Offs(pOrigin,133.15,253.06,6.00),v60,z5,tPen\WObj:=wPaper;
    MoveL Offs(pOrigin,136.51,259.76,6.00),vTravel,z5,tPen\WObj:=wPaper;
    MoveL Offs(pOrigin,136.51,259.76,0.00),v60,z0,tPen\WObj:=wPaper;
    MoveL Offs(pOrigin,136.99,260.24,0.00),v40,z0,tPen\WObj:=wPaper;
    MoveL Offs(pOrigin,136.99,260.72,0.00),v40,z0,tPen\WObj:=wPaper;
    MoveL Offs(pOrigin,136.51,259.76,0.00),v40,z0,tPen\WObj:=wPaper;
    MoveL Offs(pOrigin,136.99,260.24,0.00),v40,z0,tPen\WObj:=wPaper;
    MoveL Offs(pOrigin,136.99,260.72,0.00),v40,z0,tPen\WObj:=wPaper;
    MoveL Offs(pOrigin,136.51,259.76,0.00),v40,fine,tPen\WObj:=wPaper;
    MoveL Offs(pOrigin,136.51,259.76,6.00),v60,z5,tPen\WObj:=wPaper;
    MoveL Offs(pOrigin,139.86,265.03,6.00),vTravel,z5,tPen\WObj:=wPaper;
    MoveL Offs(pOrigin,139.86,265.03,0.00),v60,z0,tPen\WObj:=wPaper;
    MoveL Offs(pOrigin,140.34,265.51,0.00),v40,z0,tPen\WObj:=wPaper;
    MoveL Offs(pOrigin,140.34,265.99,0.00),v40,z0,tPen\WObj:=wPaper;
    MoveL Offs(pOrigin,139.86,265.03,0.00),v40,z0,tPen\WObj:=wPaper;
    MoveL Offs(pOrigin,140.34,265.51,0.00),v40,z0,tPen\WObj:=wPaper;
    MoveL Offs(pOrigin,140.34,265.99,0.00),v40,z0,tPen\WObj:=wPaper;
    MoveL Offs(pOrigin,139.86,265.03,0.00),v40,fine,tPen\WObj:=wPaper;
    MoveL Offs(pOrigin,139.86,265.03,6.00),v60,z5,tPen\WObj:=wPaper;
    MoveL Offs(pOrigin,140.82,266.46,6.00),vTravel,z5,tPen\WObj:=wPaper;
    MoveL Offs(pOrigin,140.82,266.46,0.00),v60,z0,tPen\WObj:=wPaper;
    MoveL Offs(pOrigin,141.30,266.94,0.00),v40,z0,tPen\WObj:=wPaper;
    MoveL Offs(pOrigin,141.30,267.42,0.00),v40,z0,tPen\WObj:=wPaper;
    MoveL Offs(pOrigin,140.82,266.46,0.00),v40,z0,tPen\WObj:=wPaper;
    MoveL Offs(pOrigin,141.30,266.94,0.00),v40,z0,tPen\WObj:=wPaper;
    MoveL Offs(pOrigin,141.30,267.42,0.00),v40,z0,tPen\WObj:=wPaper;
    MoveL Offs(pOrigin,140.82,266.46,0.00),v40,fine,tPen\WObj:=wPaper;
    MoveL Offs(pOrigin,140.82,266.46,6.00),v60,z5,tPen\WObj:=wPaper;
  ENDPROC

  PROC DrawPart38()
    MoveL Offs(pOrigin,141.77,268.38,6.00),vTravel,z5,tPen\WObj:=wPaper;
    MoveL Offs(pOrigin,141.77,268.38,0.00),v60,z0,tPen\WObj:=wPaper;
    MoveL Offs(pOrigin,142.73,269.34,0.00),v40,z0,tPen\WObj:=wPaper;
    MoveL Offs(pOrigin,141.77,268.38,0.00),v40,fine,tPen\WObj:=wPaper;
    MoveL Offs(pOrigin,141.77,268.38,6.00),v60,z5,tPen\WObj:=wPaper;
    MoveL Offs(pOrigin,143.21,269.82,6.00),vTravel,z5,tPen\WObj:=wPaper;
    MoveL Offs(pOrigin,143.21,269.82,0.00),v60,z0,tPen\WObj:=wPaper;
    MoveL Offs(pOrigin,144.65,271.73,0.00),v40,z0,tPen\WObj:=wPaper;
    MoveL Offs(pOrigin,143.21,269.82,0.00),v40,fine,tPen\WObj:=wPaper;
    MoveL Offs(pOrigin,143.21,269.82,6.00),v60,z5,tPen\WObj:=wPaper;
    MoveL Offs(pOrigin,145.13,272.69,6.00),vTravel,z5,tPen\WObj:=wPaper;
    MoveL Offs(pOrigin,145.13,272.69,0.00),v60,z0,tPen\WObj:=wPaper;
    MoveL Offs(pOrigin,146.08,273.65,0.00),v40,z0,tPen\WObj:=wPaper;
    MoveL Offs(pOrigin,145.13,272.69,0.00),v40,fine,tPen\WObj:=wPaper;
    MoveL Offs(pOrigin,145.13,272.69,6.00),v60,z5,tPen\WObj:=wPaper;
    MoveL Offs(pOrigin,147.52,275.56,6.00),vTravel,z5,tPen\WObj:=wPaper;
    MoveL Offs(pOrigin,147.52,275.56,0.00),v60,z0,tPen\WObj:=wPaper;
    MoveL Offs(pOrigin,148.48,276.52,0.00),v40,z0,tPen\WObj:=wPaper;
    MoveL Offs(pOrigin,147.52,275.56,0.00),v40,fine,tPen\WObj:=wPaper;
    MoveL Offs(pOrigin,147.52,275.56,6.00),v60,z5,tPen\WObj:=wPaper;
    MoveL Offs(pOrigin,149.92,278.44,6.00),vTravel,z5,tPen\WObj:=wPaper;
    MoveL Offs(pOrigin,149.92,278.44,0.00),v60,z0,tPen\WObj:=wPaper;
    MoveL Offs(pOrigin,151.35,279.87,0.00),v40,z0,tPen\WObj:=wPaper;
    MoveL Offs(pOrigin,149.92,278.44,0.00),v40,fine,tPen\WObj:=wPaper;
    MoveL Offs(pOrigin,149.92,278.44,6.00),v60,z5,tPen\WObj:=wPaper;
    MoveL Offs(pOrigin,152.31,281.31,6.00),vTravel,z5,tPen\WObj:=wPaper;
    MoveL Offs(pOrigin,152.31,281.31,0.00),v60,z0,tPen\WObj:=wPaper;
    MoveL Offs(pOrigin,157.10,286.10,0.00),v40,z0,tPen\WObj:=wPaper;
    MoveL Offs(pOrigin,152.31,281.31,0.00),v40,fine,tPen\WObj:=wPaper;
    MoveL Offs(pOrigin,152.31,281.31,6.00),v60,z5,tPen\WObj:=wPaper;
    MoveL Offs(pOrigin,157.58,286.58,6.00),vTravel,z5,tPen\WObj:=wPaper;
    MoveL Offs(pOrigin,157.58,286.58,0.00),v60,z0,tPen\WObj:=wPaper;
    MoveL Offs(pOrigin,161.41,290.41,0.00),v40,z0,tPen\WObj:=wPaper;
    MoveL Offs(pOrigin,157.58,286.58,0.00),v40,fine,tPen\WObj:=wPaper;
    MoveL Offs(pOrigin,157.58,286.58,6.00),v60,z5,tPen\WObj:=wPaper;
    MoveL Offs(pOrigin,162.37,290.89,6.00),vTravel,z5,tPen\WObj:=wPaper;
    MoveL Offs(pOrigin,162.37,290.89,0.00),v60,z0,tPen\WObj:=wPaper;
    MoveL Offs(pOrigin,164.76,293.28,0.00),v40,z0,tPen\WObj:=wPaper;
    MoveL Offs(pOrigin,162.37,290.89,0.00),v40,fine,tPen\WObj:=wPaper;
    MoveL Offs(pOrigin,162.37,290.89,6.00),v60,z5,tPen\WObj:=wPaper;
    MoveL Offs(pOrigin,165.72,293.76,6.00),vTravel,z5,tPen\WObj:=wPaper;
    MoveL Offs(pOrigin,165.72,293.76,0.00),v60,z0,tPen\WObj:=wPaper;
    MoveL Offs(pOrigin,168.59,296.63,0.00),v40,z0,tPen\WObj:=wPaper;
    MoveL Offs(pOrigin,165.72,293.76,0.00),v40,fine,tPen\WObj:=wPaper;
    MoveL Offs(pOrigin,165.72,293.76,6.00),v60,z5,tPen\WObj:=wPaper;
    MoveL Offs(pOrigin,170.03,297.59,6.00),vTravel,z5,tPen\WObj:=wPaper;
    MoveL Offs(pOrigin,170.03,297.59,0.00),v60,z0,tPen\WObj:=wPaper;
    MoveL Offs(pOrigin,170.51,297.59,0.00),v40,z0,tPen\WObj:=wPaper;
    MoveL Offs(pOrigin,171.46,298.55,0.00),v40,z0,tPen\WObj:=wPaper;
    MoveL Offs(pOrigin,170.03,297.59,0.00),v40,z0,tPen\WObj:=wPaper;
    MoveL Offs(pOrigin,170.51,297.59,0.00),v40,z0,tPen\WObj:=wPaper;
    MoveL Offs(pOrigin,171.46,298.55,0.00),v40,z0,tPen\WObj:=wPaper;
    MoveL Offs(pOrigin,170.03,297.59,0.00),v40,fine,tPen\WObj:=wPaper;
    MoveL Offs(pOrigin,170.03,297.59,6.00),v60,z5,tPen\WObj:=wPaper;
    MoveL Offs(pOrigin,175.77,301.42,6.00),vTravel,z5,tPen\WObj:=wPaper;
    MoveL Offs(pOrigin,175.77,301.42,0.00),v60,z0,tPen\WObj:=wPaper;
    MoveL Offs(pOrigin,176.25,301.42,0.00),v40,z0,tPen\WObj:=wPaper;
    MoveL Offs(pOrigin,177.21,302.38,0.00),v40,z0,tPen\WObj:=wPaper;
    MoveL Offs(pOrigin,175.77,301.42,0.00),v40,z0,tPen\WObj:=wPaper;
    MoveL Offs(pOrigin,176.25,301.42,0.00),v40,z0,tPen\WObj:=wPaper;
    MoveL Offs(pOrigin,177.21,302.38,0.00),v40,z0,tPen\WObj:=wPaper;
    MoveL Offs(pOrigin,175.77,301.42,0.00),v40,fine,tPen\WObj:=wPaper;
    MoveL Offs(pOrigin,175.77,301.42,6.00),v60,z5,tPen\WObj:=wPaper;
    MoveL Offs(pOrigin,178.65,303.34,6.00),vTravel,z5,tPen\WObj:=wPaper;
    MoveL Offs(pOrigin,178.65,303.34,0.00),v60,z0,tPen\WObj:=wPaper;
    MoveL Offs(pOrigin,179.13,303.34,0.00),v40,z0,tPen\WObj:=wPaper;
    MoveL Offs(pOrigin,179.61,303.82,0.00),v40,z0,tPen\WObj:=wPaper;
    MoveL Offs(pOrigin,178.65,303.34,0.00),v40,z0,tPen\WObj:=wPaper;
    MoveL Offs(pOrigin,179.13,303.34,0.00),v40,z0,tPen\WObj:=wPaper;
    MoveL Offs(pOrigin,179.61,303.82,0.00),v40,z0,tPen\WObj:=wPaper;
    MoveL Offs(pOrigin,178.65,303.34,0.00),v40,fine,tPen\WObj:=wPaper;
    MoveL Offs(pOrigin,178.65,303.34,6.00),v60,z5,tPen\WObj:=wPaper;
    MoveL Offs(pOrigin,182.48,305.73,6.00),vTravel,z5,tPen\WObj:=wPaper;
    MoveL Offs(pOrigin,182.48,305.73,0.00),v60,z0,tPen\WObj:=wPaper;
    MoveL Offs(pOrigin,182.96,305.73,0.00),v40,z0,tPen\WObj:=wPaper;
    MoveL Offs(pOrigin,183.44,306.21,0.00),v40,z0,tPen\WObj:=wPaper;
    MoveL Offs(pOrigin,182.48,305.73,0.00),v40,z0,tPen\WObj:=wPaper;
    MoveL Offs(pOrigin,182.96,305.73,0.00),v40,z0,tPen\WObj:=wPaper;
    MoveL Offs(pOrigin,183.44,306.21,0.00),v40,z0,tPen\WObj:=wPaper;
    MoveL Offs(pOrigin,182.48,305.73,0.00),v40,fine,tPen\WObj:=wPaper;
    MoveL Offs(pOrigin,182.48,305.73,6.00),v60,z5,tPen\WObj:=wPaper;
    MoveL Offs(pOrigin,186.79,308.13,6.00),vTravel,z5,tPen\WObj:=wPaper;
    MoveL Offs(pOrigin,186.79,308.13,0.00),v60,z0,tPen\WObj:=wPaper;
    MoveL Offs(pOrigin,187.27,308.13,0.00),v40,z0,tPen\WObj:=wPaper;
    MoveL Offs(pOrigin,187.75,308.61,0.00),v40,z0,tPen\WObj:=wPaper;
    MoveL Offs(pOrigin,186.79,308.13,0.00),v40,z0,tPen\WObj:=wPaper;
    MoveL Offs(pOrigin,187.27,308.13,0.00),v40,z0,tPen\WObj:=wPaper;
    MoveL Offs(pOrigin,187.75,308.61,0.00),v40,z0,tPen\WObj:=wPaper;
    MoveL Offs(pOrigin,186.79,308.13,0.00),v40,fine,tPen\WObj:=wPaper;
    MoveL Offs(pOrigin,186.79,308.13,6.00),v60,z5,tPen\WObj:=wPaper;
    MoveL Offs(pOrigin,189.66,300.46,6.00),vTravel,z5,tPen\WObj:=wPaper;
    MoveL Offs(pOrigin,189.66,300.46,0.00),v60,z0,tPen\WObj:=wPaper;
    MoveL Offs(pOrigin,190.14,300.46,0.00),v40,z0,tPen\WObj:=wPaper;
    MoveL Offs(pOrigin,189.66,299.99,0.00),v40,z0,tPen\WObj:=wPaper;
    MoveL Offs(pOrigin,189.66,300.46,0.00),v40,z0,tPen\WObj:=wPaper;
    MoveL Offs(pOrigin,190.14,300.46,0.00),v40,z0,tPen\WObj:=wPaper;
    MoveL Offs(pOrigin,189.66,299.99,0.00),v40,z0,tPen\WObj:=wPaper;
    MoveL Offs(pOrigin,189.66,300.46,0.00),v40,fine,tPen\WObj:=wPaper;
    MoveL Offs(pOrigin,189.66,300.46,6.00),v60,z5,tPen\WObj:=wPaper;
    MoveL Offs(pOrigin,191.58,300.94,6.00),vTravel,z5,tPen\WObj:=wPaper;
    MoveL Offs(pOrigin,191.58,300.94,0.00),v60,z0,tPen\WObj:=wPaper;
    MoveL Offs(pOrigin,191.58,301.42,0.00),v40,z0,tPen\WObj:=wPaper;
    MoveL Offs(pOrigin,192.06,301.42,0.00),v40,z0,tPen\WObj:=wPaper;
    MoveL Offs(pOrigin,191.58,300.94,0.00),v40,z0,tPen\WObj:=wPaper;
    MoveL Offs(pOrigin,191.58,301.42,0.00),v40,z0,tPen\WObj:=wPaper;
    MoveL Offs(pOrigin,192.06,301.42,0.00),v40,z0,tPen\WObj:=wPaper;
    MoveL Offs(pOrigin,191.58,300.94,0.00),v40,fine,tPen\WObj:=wPaper;
    MoveL Offs(pOrigin,191.58,300.94,6.00),v60,z5,tPen\WObj:=wPaper;
    MoveL Offs(pOrigin,185.83,298.07,6.00),vTravel,z5,tPen\WObj:=wPaper;
    MoveL Offs(pOrigin,185.83,298.07,0.00),v60,z0,tPen\WObj:=wPaper;
    MoveL Offs(pOrigin,185.35,297.59,0.00),v40,z0,tPen\WObj:=wPaper;
    MoveL Offs(pOrigin,185.35,298.07,0.00),v40,z0,tPen\WObj:=wPaper;
    MoveL Offs(pOrigin,185.83,298.07,0.00),v40,z0,tPen\WObj:=wPaper;
    MoveL Offs(pOrigin,185.35,297.59,0.00),v40,z0,tPen\WObj:=wPaper;
    MoveL Offs(pOrigin,185.35,298.07,0.00),v40,z0,tPen\WObj:=wPaper;
    MoveL Offs(pOrigin,185.83,298.07,0.00),v40,fine,tPen\WObj:=wPaper;
    MoveL Offs(pOrigin,185.83,298.07,6.00),v60,z5,tPen\WObj:=wPaper;
    MoveL Offs(pOrigin,164.76,266.94,6.00),vTravel,z5,tPen\WObj:=wPaper;
    MoveL Offs(pOrigin,164.76,266.94,0.00),v60,z0,tPen\WObj:=wPaper;
    MoveL Offs(pOrigin,161.89,264.07,0.00),v40,z0,tPen\WObj:=wPaper;
  ENDPROC

  PROC DrawPart39()
    MoveL Offs(pOrigin,161.89,264.55,0.00),v40,z0,tPen\WObj:=wPaper;
    MoveL Offs(pOrigin,162.37,264.55,0.00),v40,z0,tPen\WObj:=wPaper;
    MoveL Offs(pOrigin,164.76,266.94,0.00),v40,z0,tPen\WObj:=wPaper;
    MoveL Offs(pOrigin,161.89,264.07,0.00),v40,z0,tPen\WObj:=wPaper;
    MoveL Offs(pOrigin,161.89,264.55,0.00),v40,z0,tPen\WObj:=wPaper;
    MoveL Offs(pOrigin,162.37,264.55,0.00),v40,z0,tPen\WObj:=wPaper;
    MoveL Offs(pOrigin,164.76,266.94,0.00),v40,fine,tPen\WObj:=wPaper;
    MoveL Offs(pOrigin,164.76,266.94,6.00),v60,z5,tPen\WObj:=wPaper;
    MoveL Offs(pOrigin,169.07,261.20,6.00),vTravel,z5,tPen\WObj:=wPaper;
    MoveL Offs(pOrigin,169.07,261.20,0.00),v60,z0,tPen\WObj:=wPaper;
    MoveL Offs(pOrigin,170.03,262.15,0.00),v40,z0,tPen\WObj:=wPaper;
    MoveL Offs(pOrigin,169.07,261.20,0.00),v40,fine,tPen\WObj:=wPaper;
    MoveL Offs(pOrigin,169.07,261.20,6.00),v60,z5,tPen\WObj:=wPaper;
    MoveL Offs(pOrigin,170.51,262.63,6.00),vTravel,z5,tPen\WObj:=wPaper;
    MoveL Offs(pOrigin,170.51,262.63,0.00),v60,z0,tPen\WObj:=wPaper;
    MoveL Offs(pOrigin,175.30,267.42,0.00),v40,z0,tPen\WObj:=wPaper;
    MoveL Offs(pOrigin,170.51,262.63,0.00),v40,fine,tPen\WObj:=wPaper;
    MoveL Offs(pOrigin,170.51,262.63,6.00),v60,z5,tPen\WObj:=wPaper;
    MoveL Offs(pOrigin,165.72,257.85,6.00),vTravel,z5,tPen\WObj:=wPaper;
    MoveL Offs(pOrigin,165.72,257.85,0.00),v60,z0,tPen\WObj:=wPaper;
    MoveL Offs(pOrigin,168.11,260.24,0.00),v40,z0,tPen\WObj:=wPaper;
    MoveL Offs(pOrigin,165.72,257.85,0.00),v40,fine,tPen\WObj:=wPaper;
    MoveL Offs(pOrigin,165.72,257.85,6.00),v60,z5,tPen\WObj:=wPaper;
    MoveL Offs(pOrigin,163.80,255.45,6.00),vTravel,z5,tPen\WObj:=wPaper;
    MoveL Offs(pOrigin,163.80,255.45,0.00),v60,z0,tPen\WObj:=wPaper;
    MoveL Offs(pOrigin,165.24,256.89,0.00),v40,z0,tPen\WObj:=wPaper;
    MoveL Offs(pOrigin,163.80,255.45,0.00),v40,fine,tPen\WObj:=wPaper;
    MoveL Offs(pOrigin,163.80,255.45,6.00),v60,z5,tPen\WObj:=wPaper;
    MoveL Offs(pOrigin,160.45,251.14,6.00),vTravel,z5,tPen\WObj:=wPaper;
    MoveL Offs(pOrigin,160.45,251.14,0.00),v60,z0,tPen\WObj:=wPaper;
    MoveL Offs(pOrigin,159.97,250.18,0.00),v40,z0,tPen\WObj:=wPaper;
    MoveL Offs(pOrigin,160.45,250.66,0.00),v40,z0,tPen\WObj:=wPaper;
    MoveL Offs(pOrigin,160.45,251.14,0.00),v40,z0,tPen\WObj:=wPaper;
    MoveL Offs(pOrigin,159.97,250.18,0.00),v40,z0,tPen\WObj:=wPaper;
    MoveL Offs(pOrigin,160.45,250.66,0.00),v40,z0,tPen\WObj:=wPaper;
    MoveL Offs(pOrigin,160.45,251.14,0.00),v40,fine,tPen\WObj:=wPaper;
    MoveL Offs(pOrigin,160.45,251.14,6.00),v60,z5,tPen\WObj:=wPaper;
    MoveL Offs(pOrigin,158.06,247.31,6.00),vTravel,z5,tPen\WObj:=wPaper;
    MoveL Offs(pOrigin,158.06,247.31,0.00),v60,z0,tPen\WObj:=wPaper;
    MoveL Offs(pOrigin,159.01,248.75,0.00),v40,z0,tPen\WObj:=wPaper;
    MoveL Offs(pOrigin,158.06,247.31,0.00),v40,fine,tPen\WObj:=wPaper;
    MoveL Offs(pOrigin,158.06,247.31,6.00),v60,z5,tPen\WObj:=wPaper;
    MoveL Offs(pOrigin,155.66,244.44,6.00),vTravel,z5,tPen\WObj:=wPaper;
    MoveL Offs(pOrigin,155.66,244.44,0.00),v60,z0,tPen\WObj:=wPaper;
    MoveL Offs(pOrigin,156.62,245.39,0.00),v40,z0,tPen\WObj:=wPaper;
    MoveL Offs(pOrigin,155.66,244.44,0.00),v40,fine,tPen\WObj:=wPaper;
    MoveL Offs(pOrigin,155.66,244.44,6.00),v60,z5,tPen\WObj:=wPaper;
    MoveL Offs(pOrigin,149.92,245.39,6.00),vTravel,z5,tPen\WObj:=wPaper;
    MoveL Offs(pOrigin,149.92,245.39,0.00),v60,z0,tPen\WObj:=wPaper;
    MoveL Offs(pOrigin,149.44,244.44,0.00),v40,z0,tPen\WObj:=wPaper;
    MoveL Offs(pOrigin,149.44,244.92,0.00),v40,z0,tPen\WObj:=wPaper;
    MoveL Offs(pOrigin,149.92,245.39,0.00),v40,z0,tPen\WObj:=wPaper;
    MoveL Offs(pOrigin,149.44,244.44,0.00),v40,z0,tPen\WObj:=wPaper;
    MoveL Offs(pOrigin,149.44,244.92,0.00),v40,z0,tPen\WObj:=wPaper;
    MoveL Offs(pOrigin,149.92,245.39,0.00),v40,fine,tPen\WObj:=wPaper;
    MoveL Offs(pOrigin,149.92,245.39,6.00),v60,z5,tPen\WObj:=wPaper;
    MoveL Offs(pOrigin,151.83,249.23,6.00),vTravel,z5,tPen\WObj:=wPaper;
    MoveL Offs(pOrigin,151.83,249.23,0.00),v60,z0,tPen\WObj:=wPaper;
    MoveL Offs(pOrigin,151.83,249.70,0.00),v40,z0,tPen\WObj:=wPaper;
    MoveL Offs(pOrigin,152.31,250.18,0.00),v40,z0,tPen\WObj:=wPaper;
    MoveL Offs(pOrigin,151.83,249.23,0.00),v40,z0,tPen\WObj:=wPaper;
    MoveL Offs(pOrigin,151.83,249.70,0.00),v40,z0,tPen\WObj:=wPaper;
    MoveL Offs(pOrigin,152.31,250.18,0.00),v40,z0,tPen\WObj:=wPaper;
    MoveL Offs(pOrigin,151.83,249.23,0.00),v40,fine,tPen\WObj:=wPaper;
    MoveL Offs(pOrigin,151.83,249.23,6.00),v60,z5,tPen\WObj:=wPaper;
    MoveL Offs(pOrigin,153.75,252.58,6.00),vTravel,z5,tPen\WObj:=wPaper;
    MoveL Offs(pOrigin,153.75,252.58,0.00),v60,z0,tPen\WObj:=wPaper;
    MoveL Offs(pOrigin,153.75,253.06,0.00),v40,z0,tPen\WObj:=wPaper;
    MoveL Offs(pOrigin,154.70,254.01,0.00),v40,z0,tPen\WObj:=wPaper;
    MoveL Offs(pOrigin,153.75,252.58,0.00),v40,z0,tPen\WObj:=wPaper;
    MoveL Offs(pOrigin,153.75,253.06,0.00),v40,z0,tPen\WObj:=wPaper;
    MoveL Offs(pOrigin,154.70,254.01,0.00),v40,z0,tPen\WObj:=wPaper;
    MoveL Offs(pOrigin,153.75,252.58,0.00),v40,fine,tPen\WObj:=wPaper;
    MoveL Offs(pOrigin,153.75,252.58,6.00),v60,z5,tPen\WObj:=wPaper;
    MoveL Offs(pOrigin,156.14,256.41,6.00),vTravel,z5,tPen\WObj:=wPaper;
    MoveL Offs(pOrigin,156.14,256.41,0.00),v60,z0,tPen\WObj:=wPaper;
    MoveL Offs(pOrigin,156.14,256.89,0.00),v40,z0,tPen\WObj:=wPaper;
    MoveL Offs(pOrigin,156.62,256.89,0.00),v40,z0,tPen\WObj:=wPaper;
    MoveL Offs(pOrigin,156.14,256.41,0.00),v40,z0,tPen\WObj:=wPaper;
    MoveL Offs(pOrigin,156.14,256.89,0.00),v40,z0,tPen\WObj:=wPaper;
    MoveL Offs(pOrigin,156.62,256.89,0.00),v40,z0,tPen\WObj:=wPaper;
    MoveL Offs(pOrigin,156.14,256.41,0.00),v40,fine,tPen\WObj:=wPaper;
    MoveL Offs(pOrigin,156.14,256.41,6.00),v60,z5,tPen\WObj:=wPaper;
    MoveL Offs(pOrigin,159.01,260.24,6.00),vTravel,z5,tPen\WObj:=wPaper;
    MoveL Offs(pOrigin,159.01,260.24,0.00),v60,z0,tPen\WObj:=wPaper;
    MoveL Offs(pOrigin,159.01,260.72,0.00),v40,z0,tPen\WObj:=wPaper;
    MoveL Offs(pOrigin,159.49,260.72,0.00),v40,z0,tPen\WObj:=wPaper;
    MoveL Offs(pOrigin,159.97,261.20,0.00),v40,z0,tPen\WObj:=wPaper;
    MoveL Offs(pOrigin,159.01,260.24,0.00),v40,z0,tPen\WObj:=wPaper;
    MoveL Offs(pOrigin,159.01,260.72,0.00),v40,z0,tPen\WObj:=wPaper;
    MoveL Offs(pOrigin,159.49,260.72,0.00),v40,z0,tPen\WObj:=wPaper;
    MoveL Offs(pOrigin,159.97,261.20,0.00),v40,z0,tPen\WObj:=wPaper;
    MoveL Offs(pOrigin,159.01,260.24,0.00),v40,fine,tPen\WObj:=wPaper;
    MoveL Offs(pOrigin,159.01,260.24,6.00),v60,z5,tPen\WObj:=wPaper;
    MoveL Offs(pOrigin,172.42,238.69,6.00),vTravel,z5,tPen\WObj:=wPaper;
    MoveL Offs(pOrigin,172.42,238.69,0.00),v60,z0,tPen\WObj:=wPaper;
    MoveL Offs(pOrigin,170.99,237.73,0.00),v40,z0,tPen\WObj:=wPaper;
    MoveL Offs(pOrigin,171.46,237.73,0.00),v40,z0,tPen\WObj:=wPaper;
    MoveL Offs(pOrigin,172.42,238.69,0.00),v40,z0,tPen\WObj:=wPaper;
    MoveL Offs(pOrigin,170.99,237.73,0.00),v40,z0,tPen\WObj:=wPaper;
    MoveL Offs(pOrigin,171.46,237.73,0.00),v40,z0,tPen\WObj:=wPaper;
    MoveL Offs(pOrigin,172.42,238.69,0.00),v40,z0,tPen\WObj:=wPaper;
    MoveL Offs(pOrigin,173.38,239.17,0.00),v40,z0,tPen\WObj:=wPaper;
    MoveL Offs(pOrigin,173.86,239.17,0.00),v40,z0,tPen\WObj:=wPaper;
    MoveL Offs(pOrigin,174.34,239.65,0.00),v40,z0,tPen\WObj:=wPaper;
    MoveL Offs(pOrigin,173.38,239.17,0.00),v40,z0,tPen\WObj:=wPaper;
    MoveL Offs(pOrigin,173.86,239.17,0.00),v40,z0,tPen\WObj:=wPaper;
    MoveL Offs(pOrigin,174.34,239.65,0.00),v40,z0,tPen\WObj:=wPaper;
    MoveL Offs(pOrigin,173.38,239.17,0.00),v40,fine,tPen\WObj:=wPaper;
    MoveL Offs(pOrigin,173.38,239.17,6.00),v60,z5,tPen\WObj:=wPaper;
    MoveL Offs(pOrigin,174.82,240.13,6.00),vTravel,z5,tPen\WObj:=wPaper;
    MoveL Offs(pOrigin,174.82,240.13,0.00),v60,z0,tPen\WObj:=wPaper;
    MoveL Offs(pOrigin,175.30,240.13,0.00),v40,z0,tPen\WObj:=wPaper;
    MoveL Offs(pOrigin,175.77,240.61,0.00),v40,z0,tPen\WObj:=wPaper;
    MoveL Offs(pOrigin,174.82,240.13,0.00),v40,z0,tPen\WObj:=wPaper;
    MoveL Offs(pOrigin,175.30,240.13,0.00),v40,z0,tPen\WObj:=wPaper;
    MoveL Offs(pOrigin,175.77,240.61,0.00),v40,z0,tPen\WObj:=wPaper;
    MoveL Offs(pOrigin,174.82,240.13,0.00),v40,fine,tPen\WObj:=wPaper;
    MoveL Offs(pOrigin,174.82,240.13,6.00),v60,z5,tPen\WObj:=wPaper;
    MoveL Offs(pOrigin,180.56,243.00,6.00),vTravel,z5,tPen\WObj:=wPaper;
  ENDPROC

  PROC DrawPart40()
    MoveL Offs(pOrigin,180.56,243.00,0.00),v60,z0,tPen\WObj:=wPaper;
    MoveL Offs(pOrigin,181.04,243.00,0.00),v40,z0,tPen\WObj:=wPaper;
    MoveL Offs(pOrigin,181.52,243.48,0.00),v40,z0,tPen\WObj:=wPaper;
    MoveL Offs(pOrigin,180.56,243.00,0.00),v40,z0,tPen\WObj:=wPaper;
    MoveL Offs(pOrigin,181.04,243.00,0.00),v40,z0,tPen\WObj:=wPaper;
    MoveL Offs(pOrigin,181.52,243.48,0.00),v40,z0,tPen\WObj:=wPaper;
    MoveL Offs(pOrigin,180.56,243.00,0.00),v40,fine,tPen\WObj:=wPaper;
    MoveL Offs(pOrigin,180.56,243.00,6.00),v60,z5,tPen\WObj:=wPaper;
    MoveL Offs(pOrigin,182.48,243.96,6.00),vTravel,z5,tPen\WObj:=wPaper;
    MoveL Offs(pOrigin,182.48,243.96,0.00),v60,z0,tPen\WObj:=wPaper;
    MoveL Offs(pOrigin,182.96,243.96,0.00),v40,z0,tPen\WObj:=wPaper;
    MoveL Offs(pOrigin,183.44,244.44,0.00),v40,z0,tPen\WObj:=wPaper;
    MoveL Offs(pOrigin,182.48,243.96,0.00),v40,z0,tPen\WObj:=wPaper;
    MoveL Offs(pOrigin,182.96,243.96,0.00),v40,z0,tPen\WObj:=wPaper;
    MoveL Offs(pOrigin,183.44,244.44,0.00),v40,z0,tPen\WObj:=wPaper;
    MoveL Offs(pOrigin,182.48,243.96,0.00),v40,fine,tPen\WObj:=wPaper;
    MoveL Offs(pOrigin,182.48,243.96,6.00),v60,z5,tPen\WObj:=wPaper;
    MoveL Offs(pOrigin,185.35,245.39,6.00),vTravel,z5,tPen\WObj:=wPaper;
    MoveL Offs(pOrigin,185.35,245.39,0.00),v60,z0,tPen\WObj:=wPaper;
    MoveL Offs(pOrigin,185.83,245.39,0.00),v40,z0,tPen\WObj:=wPaper;
    MoveL Offs(pOrigin,186.31,245.87,0.00),v40,z0,tPen\WObj:=wPaper;
    MoveL Offs(pOrigin,185.35,245.39,0.00),v40,z0,tPen\WObj:=wPaper;
    MoveL Offs(pOrigin,185.83,245.39,0.00),v40,z0,tPen\WObj:=wPaper;
    MoveL Offs(pOrigin,186.31,245.87,0.00),v40,z0,tPen\WObj:=wPaper;
    MoveL Offs(pOrigin,185.35,245.39,0.00),v40,fine,tPen\WObj:=wPaper;
    MoveL Offs(pOrigin,185.35,245.39,6.00),v60,z5,tPen\WObj:=wPaper;
    MoveL Offs(pOrigin,187.75,246.35,6.00),vTravel,z5,tPen\WObj:=wPaper;
    MoveL Offs(pOrigin,187.75,246.35,0.00),v60,z0,tPen\WObj:=wPaper;
    MoveL Offs(pOrigin,188.23,246.35,0.00),v40,z0,tPen\WObj:=wPaper;
    MoveL Offs(pOrigin,188.70,246.83,0.00),v40,z0,tPen\WObj:=wPaper;
    MoveL Offs(pOrigin,187.75,246.35,0.00),v40,z0,tPen\WObj:=wPaper;
    MoveL Offs(pOrigin,188.23,246.35,0.00),v40,z0,tPen\WObj:=wPaper;
    MoveL Offs(pOrigin,188.70,246.83,0.00),v40,z0,tPen\WObj:=wPaper;
    MoveL Offs(pOrigin,187.75,246.35,0.00),v40,fine,tPen\WObj:=wPaper;
    MoveL Offs(pOrigin,187.75,246.35,6.00),v60,z5,tPen\WObj:=wPaper;
    MoveL Offs(pOrigin,185.35,227.20,6.00),vTravel,z5,tPen\WObj:=wPaper;
    MoveL Offs(pOrigin,185.35,227.20,0.00),v60,z0,tPen\WObj:=wPaper;
    MoveL Offs(pOrigin,184.87,226.72,0.00),v40,z0,tPen\WObj:=wPaper;
    MoveL Offs(pOrigin,184.87,227.20,0.00),v40,z0,tPen\WObj:=wPaper;
    MoveL Offs(pOrigin,185.35,227.20,0.00),v40,z0,tPen\WObj:=wPaper;
    MoveL Offs(pOrigin,184.87,226.72,0.00),v40,z0,tPen\WObj:=wPaper;
    MoveL Offs(pOrigin,184.87,227.20,0.00),v40,z0,tPen\WObj:=wPaper;
    MoveL Offs(pOrigin,185.35,227.20,0.00),v40,fine,tPen\WObj:=wPaper;
    MoveL Offs(pOrigin,185.35,227.20,6.00),v60,z5,tPen\WObj:=wPaper;
    MoveL Offs(pOrigin,182.96,225.76,6.00),vTravel,z5,tPen\WObj:=wPaper;
    MoveL Offs(pOrigin,182.96,225.76,0.00),v60,z0,tPen\WObj:=wPaper;
    MoveL Offs(pOrigin,182.48,225.28,0.00),v40,z0,tPen\WObj:=wPaper;
    MoveL Offs(pOrigin,182.48,225.76,0.00),v40,z0,tPen\WObj:=wPaper;
    MoveL Offs(pOrigin,182.96,225.76,0.00),v40,z0,tPen\WObj:=wPaper;
    MoveL Offs(pOrigin,182.48,225.28,0.00),v40,z0,tPen\WObj:=wPaper;
    MoveL Offs(pOrigin,182.48,225.76,0.00),v40,z0,tPen\WObj:=wPaper;
    MoveL Offs(pOrigin,182.96,225.76,0.00),v40,fine,tPen\WObj:=wPaper;
    MoveL Offs(pOrigin,182.96,225.76,6.00),v60,z5,tPen\WObj:=wPaper;
    MoveL Offs(pOrigin,180.08,223.85,6.00),vTravel,z5,tPen\WObj:=wPaper;
    MoveL Offs(pOrigin,180.08,223.85,0.00),v60,z0,tPen\WObj:=wPaper;
    MoveL Offs(pOrigin,179.13,222.89,0.00),v40,z0,tPen\WObj:=wPaper;
    MoveL Offs(pOrigin,179.13,223.37,0.00),v40,z0,tPen\WObj:=wPaper;
    MoveL Offs(pOrigin,179.61,223.37,0.00),v40,z0,tPen\WObj:=wPaper;
    MoveL Offs(pOrigin,180.08,223.85,0.00),v40,z0,tPen\WObj:=wPaper;
    MoveL Offs(pOrigin,179.13,222.89,0.00),v40,z0,tPen\WObj:=wPaper;
    MoveL Offs(pOrigin,179.13,223.37,0.00),v40,z0,tPen\WObj:=wPaper;
    MoveL Offs(pOrigin,179.61,223.37,0.00),v40,z0,tPen\WObj:=wPaper;
    MoveL Offs(pOrigin,180.08,223.85,0.00),v40,fine,tPen\WObj:=wPaper;
    MoveL Offs(pOrigin,180.08,223.85,6.00),v60,z5,tPen\WObj:=wPaper;
    MoveL Offs(pOrigin,177.21,221.45,6.00),vTravel,z5,tPen\WObj:=wPaper;
    MoveL Offs(pOrigin,177.21,221.45,0.00),v60,z0,tPen\WObj:=wPaper;
    MoveL Offs(pOrigin,175.77,220.01,0.00),v40,z0,tPen\WObj:=wPaper;
    MoveL Offs(pOrigin,175.77,220.49,0.00),v40,z0,tPen\WObj:=wPaper;
    MoveL Offs(pOrigin,176.25,220.49,0.00),v40,z0,tPen\WObj:=wPaper;
    MoveL Offs(pOrigin,177.21,221.45,0.00),v40,z0,tPen\WObj:=wPaper;
    MoveL Offs(pOrigin,175.77,220.01,0.00),v40,z0,tPen\WObj:=wPaper;
    MoveL Offs(pOrigin,175.77,220.49,0.00),v40,z0,tPen\WObj:=wPaper;
    MoveL Offs(pOrigin,176.25,220.49,0.00),v40,z0,tPen\WObj:=wPaper;
    MoveL Offs(pOrigin,177.21,221.45,0.00),v40,fine,tPen\WObj:=wPaper;
    MoveL Offs(pOrigin,177.21,221.45,6.00),v60,z5,tPen\WObj:=wPaper;
    MoveL Offs(pOrigin,175.30,219.54,6.00),vTravel,z5,tPen\WObj:=wPaper;
    MoveL Offs(pOrigin,175.30,219.54,0.00),v60,z0,tPen\WObj:=wPaper;
    MoveL Offs(pOrigin,172.90,217.14,0.00),v40,z0,tPen\WObj:=wPaper;
    MoveL Offs(pOrigin,172.90,217.62,0.00),v40,z0,tPen\WObj:=wPaper;
    MoveL Offs(pOrigin,173.38,217.62,0.00),v40,z0,tPen\WObj:=wPaper;
    MoveL Offs(pOrigin,175.30,219.54,0.00),v40,z0,tPen\WObj:=wPaper;
    MoveL Offs(pOrigin,172.90,217.14,0.00),v40,z0,tPen\WObj:=wPaper;
    MoveL Offs(pOrigin,172.90,217.62,0.00),v40,z0,tPen\WObj:=wPaper;
    MoveL Offs(pOrigin,173.38,217.62,0.00),v40,z0,tPen\WObj:=wPaper;
    MoveL Offs(pOrigin,175.30,219.54,0.00),v40,fine,tPen\WObj:=wPaper;
    MoveL Offs(pOrigin,175.30,219.54,6.00),v60,z5,tPen\WObj:=wPaper;
    MoveL Offs(pOrigin,172.42,216.18,6.00),vTravel,z5,tPen\WObj:=wPaper;
    MoveL Offs(pOrigin,172.42,216.18,0.00),v60,z0,tPen\WObj:=wPaper;
    MoveL Offs(pOrigin,170.99,214.75,0.00),v40,z0,tPen\WObj:=wPaper;
    MoveL Offs(pOrigin,170.99,215.23,0.00),v40,z0,tPen\WObj:=wPaper;
    MoveL Offs(pOrigin,171.46,215.23,0.00),v40,z0,tPen\WObj:=wPaper;
    MoveL Offs(pOrigin,172.42,216.18,0.00),v40,z0,tPen\WObj:=wPaper;
    MoveL Offs(pOrigin,170.99,214.75,0.00),v40,z0,tPen\WObj:=wPaper;
    MoveL Offs(pOrigin,170.99,215.23,0.00),v40,z0,tPen\WObj:=wPaper;
    MoveL Offs(pOrigin,171.46,215.23,0.00),v40,z0,tPen\WObj:=wPaper;
    MoveL Offs(pOrigin,172.42,216.18,0.00),v40,fine,tPen\WObj:=wPaper;
    MoveL Offs(pOrigin,172.42,216.18,6.00),v60,z5,tPen\WObj:=wPaper;
    MoveL Offs(pOrigin,170.03,213.31,6.00),vTravel,z5,tPen\WObj:=wPaper;
    MoveL Offs(pOrigin,170.03,213.31,0.00),v60,z0,tPen\WObj:=wPaper;
    MoveL Offs(pOrigin,169.55,212.83,0.00),v40,z0,tPen\WObj:=wPaper;
    MoveL Offs(pOrigin,169.55,213.31,0.00),v40,z0,tPen\WObj:=wPaper;
    MoveL Offs(pOrigin,170.03,213.31,0.00),v40,z0,tPen\WObj:=wPaper;
    MoveL Offs(pOrigin,169.55,212.83,0.00),v40,z0,tPen\WObj:=wPaper;
    MoveL Offs(pOrigin,169.55,213.31,0.00),v40,z0,tPen\WObj:=wPaper;
    MoveL Offs(pOrigin,170.03,213.31,0.00),v40,fine,tPen\WObj:=wPaper;
    MoveL Offs(pOrigin,170.03,213.31,6.00),v60,z5,tPen\WObj:=wPaper;
    MoveL Offs(pOrigin,169.07,211.87,6.00),vTravel,z5,tPen\WObj:=wPaper;
    MoveL Offs(pOrigin,169.07,211.87,0.00),v60,z0,tPen\WObj:=wPaper;
    MoveL Offs(pOrigin,168.59,211.39,0.00),v40,z0,tPen\WObj:=wPaper;
    MoveL Offs(pOrigin,168.59,211.87,0.00),v40,z0,tPen\WObj:=wPaper;
    MoveL Offs(pOrigin,169.07,211.87,0.00),v40,z0,tPen\WObj:=wPaper;
    MoveL Offs(pOrigin,168.59,211.39,0.00),v40,z0,tPen\WObj:=wPaper;
    MoveL Offs(pOrigin,168.59,211.87,0.00),v40,z0,tPen\WObj:=wPaper;
    MoveL Offs(pOrigin,169.07,211.87,0.00),v40,fine,tPen\WObj:=wPaper;
    MoveL Offs(pOrigin,169.07,211.87,6.00),v60,z5,tPen\WObj:=wPaper;
    MoveL Offs(pOrigin,166.20,196.55,6.00),vTravel,z5,tPen\WObj:=wPaper;
    MoveL Offs(pOrigin,166.20,196.55,0.00),v60,z0,tPen\WObj:=wPaper;
    MoveL Offs(pOrigin,166.68,195.59,0.00),v40,z0,tPen\WObj:=wPaper;
    MoveL Offs(pOrigin,166.68,196.07,0.00),v40,z0,tPen\WObj:=wPaper;
    MoveL Offs(pOrigin,166.20,196.55,0.00),v40,z0,tPen\WObj:=wPaper;
  ENDPROC

  PROC DrawPart41()
    MoveL Offs(pOrigin,166.68,195.59,0.00),v40,z0,tPen\WObj:=wPaper;
    MoveL Offs(pOrigin,166.68,196.07,0.00),v40,z0,tPen\WObj:=wPaper;
    MoveL Offs(pOrigin,166.20,196.55,0.00),v40,fine,tPen\WObj:=wPaper;
    MoveL Offs(pOrigin,166.20,196.55,6.00),v60,z5,tPen\WObj:=wPaper;
    MoveL Offs(pOrigin,167.63,195.11,6.00),vTravel,z5,tPen\WObj:=wPaper;
    MoveL Offs(pOrigin,167.63,195.11,0.00),v60,z0,tPen\WObj:=wPaper;
    MoveL Offs(pOrigin,168.11,194.63,0.00),v40,z0,tPen\WObj:=wPaper;
    MoveL Offs(pOrigin,168.11,194.15,0.00),v40,z0,tPen\WObj:=wPaper;
    MoveL Offs(pOrigin,167.63,195.11,0.00),v40,z0,tPen\WObj:=wPaper;
    MoveL Offs(pOrigin,168.11,194.63,0.00),v40,z0,tPen\WObj:=wPaper;
    MoveL Offs(pOrigin,168.11,194.15,0.00),v40,z0,tPen\WObj:=wPaper;
    MoveL Offs(pOrigin,167.63,195.11,0.00),v40,fine,tPen\WObj:=wPaper;
    MoveL Offs(pOrigin,167.63,195.11,6.00),v60,z5,tPen\WObj:=wPaper;
    MoveL Offs(pOrigin,152.79,195.11,6.00),vTravel,z5,tPen\WObj:=wPaper;
    MoveL Offs(pOrigin,152.79,195.11,0.00),v60,z0,tPen\WObj:=wPaper;
    MoveL Offs(pOrigin,152.79,195.59,0.00),v40,z0,tPen\WObj:=wPaper;
    MoveL Offs(pOrigin,152.31,195.59,0.00),v40,z0,tPen\WObj:=wPaper;
    MoveL Offs(pOrigin,152.79,195.11,0.00),v40,z0,tPen\WObj:=wPaper;
    MoveL Offs(pOrigin,152.79,195.59,0.00),v40,z0,tPen\WObj:=wPaper;
    MoveL Offs(pOrigin,152.31,195.59,0.00),v40,z0,tPen\WObj:=wPaper;
    MoveL Offs(pOrigin,152.79,195.11,0.00),v40,fine,tPen\WObj:=wPaper;
    MoveL Offs(pOrigin,152.79,195.11,6.00),v60,z5,tPen\WObj:=wPaper;
    MoveL Offs(pOrigin,151.35,196.07,6.00),vTravel,z5,tPen\WObj:=wPaper;
    MoveL Offs(pOrigin,151.35,196.07,0.00),v60,z0,tPen\WObj:=wPaper;
    MoveL Offs(pOrigin,151.35,196.55,0.00),v40,z0,tPen\WObj:=wPaper;
    MoveL Offs(pOrigin,150.39,197.51,0.00),v40,z0,tPen\WObj:=wPaper;
    MoveL Offs(pOrigin,151.35,196.07,0.00),v40,z0,tPen\WObj:=wPaper;
    MoveL Offs(pOrigin,151.35,196.55,0.00),v40,z0,tPen\WObj:=wPaper;
    MoveL Offs(pOrigin,150.39,197.51,0.00),v40,z0,tPen\WObj:=wPaper;
    MoveL Offs(pOrigin,151.35,196.07,0.00),v40,fine,tPen\WObj:=wPaper;
    MoveL Offs(pOrigin,151.35,196.07,6.00),v60,z5,tPen\WObj:=wPaper;
    MoveL Offs(pOrigin,149.92,197.99,6.00),vTravel,z5,tPen\WObj:=wPaper;
    MoveL Offs(pOrigin,149.92,197.99,0.00),v60,z0,tPen\WObj:=wPaper;
    MoveL Offs(pOrigin,149.92,198.46,0.00),v40,z0,tPen\WObj:=wPaper;
    MoveL Offs(pOrigin,149.44,198.94,0.00),v40,z0,tPen\WObj:=wPaper;
    MoveL Offs(pOrigin,149.92,197.99,0.00),v40,z0,tPen\WObj:=wPaper;
    MoveL Offs(pOrigin,149.92,198.46,0.00),v40,z0,tPen\WObj:=wPaper;
    MoveL Offs(pOrigin,149.44,198.94,0.00),v40,z0,tPen\WObj:=wPaper;
    MoveL Offs(pOrigin,149.92,197.99,0.00),v40,fine,tPen\WObj:=wPaper;
    MoveL Offs(pOrigin,149.92,197.99,6.00),v60,z5,tPen\WObj:=wPaper;
    MoveL Offs(pOrigin,148.96,213.31,6.00),vTravel,z5,tPen\WObj:=wPaper;
    MoveL Offs(pOrigin,148.96,213.31,0.00),v60,z0,tPen\WObj:=wPaper;
    MoveL Offs(pOrigin,149.44,213.79,0.00),v40,z0,tPen\WObj:=wPaper;
    MoveL Offs(pOrigin,149.44,214.27,0.00),v40,z0,tPen\WObj:=wPaper;
    MoveL Offs(pOrigin,148.96,213.31,0.00),v40,z0,tPen\WObj:=wPaper;
    MoveL Offs(pOrigin,149.44,213.79,0.00),v40,z0,tPen\WObj:=wPaper;
    MoveL Offs(pOrigin,149.44,214.27,0.00),v40,z0,tPen\WObj:=wPaper;
    MoveL Offs(pOrigin,148.96,213.31,0.00),v40,fine,tPen\WObj:=wPaper;
    MoveL Offs(pOrigin,148.96,213.31,6.00),v60,z5,tPen\WObj:=wPaper;
    MoveL Offs(pOrigin,149.92,215.23,6.00),vTravel,z5,tPen\WObj:=wPaper;
    MoveL Offs(pOrigin,149.92,215.23,0.00),v60,z0,tPen\WObj:=wPaper;
    MoveL Offs(pOrigin,150.39,215.70,0.00),v40,z0,tPen\WObj:=wPaper;
    MoveL Offs(pOrigin,150.39,216.18,0.00),v40,z0,tPen\WObj:=wPaper;
    MoveL Offs(pOrigin,149.92,215.23,0.00),v40,z0,tPen\WObj:=wPaper;
    MoveL Offs(pOrigin,150.39,215.70,0.00),v40,z0,tPen\WObj:=wPaper;
    MoveL Offs(pOrigin,150.39,216.18,0.00),v40,z0,tPen\WObj:=wPaper;
    MoveL Offs(pOrigin,149.92,215.23,0.00),v40,fine,tPen\WObj:=wPaper;
    MoveL Offs(pOrigin,149.92,215.23,6.00),v60,z5,tPen\WObj:=wPaper;
    MoveL Offs(pOrigin,151.35,218.10,6.00),vTravel,z5,tPen\WObj:=wPaper;
    MoveL Offs(pOrigin,151.35,218.10,0.00),v60,z0,tPen\WObj:=wPaper;
    MoveL Offs(pOrigin,151.83,218.58,0.00),v40,z0,tPen\WObj:=wPaper;
    MoveL Offs(pOrigin,151.83,219.06,0.00),v40,z0,tPen\WObj:=wPaper;
    MoveL Offs(pOrigin,151.35,218.10,0.00),v40,z0,tPen\WObj:=wPaper;
    MoveL Offs(pOrigin,151.83,218.58,0.00),v40,z0,tPen\WObj:=wPaper;
    MoveL Offs(pOrigin,151.83,219.06,0.00),v40,z0,tPen\WObj:=wPaper;
    MoveL Offs(pOrigin,151.35,218.10,0.00),v40,fine,tPen\WObj:=wPaper;
    MoveL Offs(pOrigin,151.35,218.10,6.00),v60,z5,tPen\WObj:=wPaper;
    MoveL Offs(pOrigin,152.79,220.49,6.00),vTravel,z5,tPen\WObj:=wPaper;
    MoveL Offs(pOrigin,152.79,220.49,0.00),v60,z0,tPen\WObj:=wPaper;
    MoveL Offs(pOrigin,153.27,220.97,0.00),v40,z0,tPen\WObj:=wPaper;
    MoveL Offs(pOrigin,153.27,221.45,0.00),v40,z0,tPen\WObj:=wPaper;
    MoveL Offs(pOrigin,152.79,220.49,0.00),v40,z0,tPen\WObj:=wPaper;
    MoveL Offs(pOrigin,153.27,220.97,0.00),v40,z0,tPen\WObj:=wPaper;
    MoveL Offs(pOrigin,153.27,221.45,0.00),v40,z0,tPen\WObj:=wPaper;
    MoveL Offs(pOrigin,152.79,220.49,0.00),v40,fine,tPen\WObj:=wPaper;
    MoveL Offs(pOrigin,152.79,220.49,6.00),v60,z5,tPen\WObj:=wPaper;
    MoveL Offs(pOrigin,154.23,222.41,6.00),vTravel,z5,tPen\WObj:=wPaper;
    MoveL Offs(pOrigin,154.23,222.41,0.00),v60,z0,tPen\WObj:=wPaper;
    MoveL Offs(pOrigin,155.66,224.32,0.00),v40,z0,tPen\WObj:=wPaper;
    MoveL Offs(pOrigin,154.23,222.41,0.00),v40,fine,tPen\WObj:=wPaper;
    MoveL Offs(pOrigin,154.23,222.41,6.00),v60,z5,tPen\WObj:=wPaper;
    MoveL Offs(pOrigin,156.14,225.28,6.00),vTravel,z5,tPen\WObj:=wPaper;
    MoveL Offs(pOrigin,156.14,225.28,0.00),v60,z0,tPen\WObj:=wPaper;
    MoveL Offs(pOrigin,159.97,229.11,0.00),v40,z0,tPen\WObj:=wPaper;
    MoveL Offs(pOrigin,156.14,225.28,0.00),v40,fine,tPen\WObj:=wPaper;
    MoveL Offs(pOrigin,156.14,225.28,6.00),v60,z5,tPen\WObj:=wPaper;
    MoveL Offs(pOrigin,160.45,229.59,6.00),vTravel,z5,tPen\WObj:=wPaper;
    MoveL Offs(pOrigin,160.45,229.59,0.00),v60,z0,tPen\WObj:=wPaper;
    MoveL Offs(pOrigin,162.37,231.51,0.00),v40,z0,tPen\WObj:=wPaper;
    MoveL Offs(pOrigin,160.45,229.59,0.00),v40,fine,tPen\WObj:=wPaper;
    MoveL Offs(pOrigin,160.45,229.59,6.00),v60,z5,tPen\WObj:=wPaper;
    MoveL Offs(pOrigin,164.28,232.94,6.00),vTravel,z5,tPen\WObj:=wPaper;
    MoveL Offs(pOrigin,164.28,232.94,0.00),v60,z0,tPen\WObj:=wPaper;
    MoveL Offs(pOrigin,165.24,233.90,0.00),v40,z0,tPen\WObj:=wPaper;
    MoveL Offs(pOrigin,164.28,232.94,0.00),v40,fine,tPen\WObj:=wPaper;
    MoveL Offs(pOrigin,164.28,232.94,6.00),v60,z5,tPen\WObj:=wPaper;
    MoveL Offs(pOrigin,167.15,235.34,6.00),vTravel,z5,tPen\WObj:=wPaper;
    MoveL Offs(pOrigin,167.15,235.34,0.00),v60,z0,tPen\WObj:=wPaper;
    MoveL Offs(pOrigin,167.63,235.34,0.00),v40,z0,tPen\WObj:=wPaper;
    MoveL Offs(pOrigin,168.59,236.30,0.00),v40,z0,tPen\WObj:=wPaper;
    MoveL Offs(pOrigin,167.15,235.34,0.00),v40,z0,tPen\WObj:=wPaper;
    MoveL Offs(pOrigin,167.63,235.34,0.00),v40,z0,tPen\WObj:=wPaper;
    MoveL Offs(pOrigin,168.59,236.30,0.00),v40,z0,tPen\WObj:=wPaper;
    MoveL Offs(pOrigin,167.15,235.34,0.00),v40,fine,tPen\WObj:=wPaper;
    MoveL Offs(pOrigin,167.15,235.34,6.00),v60,z5,tPen\WObj:=wPaper;
    MoveL Offs(pOrigin,193.49,186.49,6.00),vTravel,z5,tPen\WObj:=wPaper;
    MoveL Offs(pOrigin,193.49,186.49,0.00),v60,z0,tPen\WObj:=wPaper;
    MoveL Offs(pOrigin,193.01,185.54,0.00),v40,z0,tPen\WObj:=wPaper;
    MoveL Offs(pOrigin,193.49,186.01,0.00),v40,z0,tPen\WObj:=wPaper;
    MoveL Offs(pOrigin,193.49,186.49,0.00),v40,z0,tPen\WObj:=wPaper;
    MoveL Offs(pOrigin,193.01,185.54,0.00),v40,z0,tPen\WObj:=wPaper;
    MoveL Offs(pOrigin,193.49,186.01,0.00),v40,z0,tPen\WObj:=wPaper;
    MoveL Offs(pOrigin,193.49,186.49,0.00),v40,fine,tPen\WObj:=wPaper;
    MoveL Offs(pOrigin,193.49,186.49,6.00),v60,z5,tPen\WObj:=wPaper;
    MoveL Offs(pOrigin,223.18,141.00,6.00),vTravel,z5,tPen\WObj:=wPaper;
    MoveL Offs(pOrigin,223.18,141.00,0.00),v60,z0,tPen\WObj:=wPaper;
    MoveL Offs(pOrigin,223.66,140.04,0.00),v40,z0,tPen\WObj:=wPaper;
    MoveL Offs(pOrigin,223.66,140.52,0.00),v40,z0,tPen\WObj:=wPaper;
    MoveL Offs(pOrigin,223.18,141.00,0.00),v40,z0,tPen\WObj:=wPaper;
    MoveL Offs(pOrigin,223.66,140.04,0.00),v40,z0,tPen\WObj:=wPaper;
  ENDPROC

  PROC DrawPart42()
    MoveL Offs(pOrigin,223.66,140.52,0.00),v40,z0,tPen\WObj:=wPaper;
    MoveL Offs(pOrigin,223.18,141.00,0.00),v40,fine,tPen\WObj:=wPaper;
    MoveL Offs(pOrigin,223.18,141.00,6.00),v60,z5,tPen\WObj:=wPaper;
    MoveL Offs(pOrigin,225.10,138.13,6.00),vTravel,z5,tPen\WObj:=wPaper;
    MoveL Offs(pOrigin,225.10,138.13,0.00),v60,z0,tPen\WObj:=wPaper;
    MoveL Offs(pOrigin,225.58,137.17,0.00),v40,z0,tPen\WObj:=wPaper;
    MoveL Offs(pOrigin,225.58,137.65,0.00),v40,z0,tPen\WObj:=wPaper;
    MoveL Offs(pOrigin,225.10,138.13,0.00),v40,z0,tPen\WObj:=wPaper;
    MoveL Offs(pOrigin,225.58,137.17,0.00),v40,z0,tPen\WObj:=wPaper;
    MoveL Offs(pOrigin,225.58,137.65,0.00),v40,z0,tPen\WObj:=wPaper;
    MoveL Offs(pOrigin,225.10,138.13,0.00),v40,fine,tPen\WObj:=wPaper;
    MoveL Offs(pOrigin,225.10,138.13,6.00),v60,z5,tPen\WObj:=wPaper;
    MoveL Offs(pOrigin,226.54,136.69,6.00),vTravel,z5,tPen\WObj:=wPaper;
    MoveL Offs(pOrigin,226.54,136.69,0.00),v60,z0,tPen\WObj:=wPaper;
    MoveL Offs(pOrigin,227.01,135.73,0.00),v40,z0,tPen\WObj:=wPaper;
    MoveL Offs(pOrigin,227.01,136.21,0.00),v40,z0,tPen\WObj:=wPaper;
    MoveL Offs(pOrigin,226.54,136.69,0.00),v40,z0,tPen\WObj:=wPaper;
    MoveL Offs(pOrigin,227.01,135.73,0.00),v40,z0,tPen\WObj:=wPaper;
    MoveL Offs(pOrigin,227.01,136.21,0.00),v40,z0,tPen\WObj:=wPaper;
    MoveL Offs(pOrigin,226.54,136.69,0.00),v40,fine,tPen\WObj:=wPaper;
    MoveL Offs(pOrigin,226.54,136.69,6.00),v60,z5,tPen\WObj:=wPaper;
    MoveL Offs(pOrigin,227.97,135.25,6.00),vTravel,z5,tPen\WObj:=wPaper;
    MoveL Offs(pOrigin,227.97,135.25,0.00),v60,z0,tPen\WObj:=wPaper;
    MoveL Offs(pOrigin,228.93,134.30,0.00),v40,z0,tPen\WObj:=wPaper;
    MoveL Offs(pOrigin,227.97,135.25,0.00),v40,fine,tPen\WObj:=wPaper;
    MoveL Offs(pOrigin,227.97,135.25,6.00),v60,z5,tPen\WObj:=wPaper;
    MoveL Offs(pOrigin,229.89,133.82,6.00),vTravel,z5,tPen\WObj:=wPaper;
    MoveL Offs(pOrigin,229.89,133.82,0.00),v60,z0,tPen\WObj:=wPaper;
    MoveL Offs(pOrigin,230.37,133.34,0.00),v40,z0,tPen\WObj:=wPaper;
    MoveL Offs(pOrigin,230.85,133.34,0.00),v40,z0,tPen\WObj:=wPaper;
    MoveL Offs(pOrigin,229.89,133.82,0.00),v40,z0,tPen\WObj:=wPaper;
    MoveL Offs(pOrigin,230.37,133.34,0.00),v40,z0,tPen\WObj:=wPaper;
    MoveL Offs(pOrigin,230.85,133.34,0.00),v40,z0,tPen\WObj:=wPaper;
    MoveL Offs(pOrigin,229.89,133.82,0.00),v40,fine,tPen\WObj:=wPaper;
    MoveL Offs(pOrigin,229.89,133.82,6.00),v60,z5,tPen\WObj:=wPaper;
    MoveL Offs(pOrigin,155.66,144.83,6.00),vTravel,z5,tPen\WObj:=wPaper;
    MoveL Offs(pOrigin,155.66,144.83,0.00),v60,z0,tPen\WObj:=wPaper;
    MoveL Offs(pOrigin,155.18,144.35,0.00),v40,z0,tPen\WObj:=wPaper;
    MoveL Offs(pOrigin,155.18,144.83,0.00),v40,z0,tPen\WObj:=wPaper;
    MoveL Offs(pOrigin,155.66,144.83,0.00),v40,z0,tPen\WObj:=wPaper;
    MoveL Offs(pOrigin,155.18,144.35,0.00),v40,z0,tPen\WObj:=wPaper;
    MoveL Offs(pOrigin,155.18,144.83,0.00),v40,z0,tPen\WObj:=wPaper;
    MoveL Offs(pOrigin,155.66,144.83,0.00),v40,fine,tPen\WObj:=wPaper;
    MoveL Offs(pOrigin,155.66,144.83,6.00),v60,z5,tPen\WObj:=wPaper;
    MoveL Offs(pOrigin,151.83,142.44,6.00),vTravel,z5,tPen\WObj:=wPaper;
    MoveL Offs(pOrigin,151.83,142.44,0.00),v60,z0,tPen\WObj:=wPaper;
    MoveL Offs(pOrigin,151.35,141.96,0.00),v40,z0,tPen\WObj:=wPaper;
    MoveL Offs(pOrigin,151.35,142.44,0.00),v40,z0,tPen\WObj:=wPaper;
    MoveL Offs(pOrigin,151.83,142.44,0.00),v40,z0,tPen\WObj:=wPaper;
    MoveL Offs(pOrigin,151.35,141.96,0.00),v40,z0,tPen\WObj:=wPaper;
    MoveL Offs(pOrigin,151.35,142.44,0.00),v40,z0,tPen\WObj:=wPaper;
    MoveL Offs(pOrigin,151.83,142.44,0.00),v40,fine,tPen\WObj:=wPaper;
    MoveL Offs(pOrigin,151.83,142.44,6.00),v60,z5,tPen\WObj:=wPaper;
    MoveL Offs(pOrigin,150.39,141.48,6.00),vTravel,z5,tPen\WObj:=wPaper;
    MoveL Offs(pOrigin,150.39,141.48,0.00),v60,z0,tPen\WObj:=wPaper;
    MoveL Offs(pOrigin,149.44,140.52,0.00),v40,z0,tPen\WObj:=wPaper;
    MoveL Offs(pOrigin,149.44,141.00,0.00),v40,z0,tPen\WObj:=wPaper;
    MoveL Offs(pOrigin,149.92,141.00,0.00),v40,z0,tPen\WObj:=wPaper;
    MoveL Offs(pOrigin,150.39,141.48,0.00),v40,z0,tPen\WObj:=wPaper;
    MoveL Offs(pOrigin,149.44,140.52,0.00),v40,z0,tPen\WObj:=wPaper;
    MoveL Offs(pOrigin,149.44,141.00,0.00),v40,z0,tPen\WObj:=wPaper;
    MoveL Offs(pOrigin,149.92,141.00,0.00),v40,z0,tPen\WObj:=wPaper;
    MoveL Offs(pOrigin,150.39,141.48,0.00),v40,fine,tPen\WObj:=wPaper;
    MoveL Offs(pOrigin,150.39,141.48,6.00),v60,z5,tPen\WObj:=wPaper;
    MoveL Offs(pOrigin,148.48,140.04,6.00),vTravel,z5,tPen\WObj:=wPaper;
    MoveL Offs(pOrigin,148.48,140.04,0.00),v60,z0,tPen\WObj:=wPaper;
    MoveL Offs(pOrigin,148.00,139.56,0.00),v40,z0,tPen\WObj:=wPaper;
    MoveL Offs(pOrigin,148.00,140.04,0.00),v40,z0,tPen\WObj:=wPaper;
    MoveL Offs(pOrigin,148.48,140.04,0.00),v40,z0,tPen\WObj:=wPaper;
    MoveL Offs(pOrigin,148.00,139.56,0.00),v40,z0,tPen\WObj:=wPaper;
    MoveL Offs(pOrigin,148.00,140.04,0.00),v40,z0,tPen\WObj:=wPaper;
    MoveL Offs(pOrigin,148.48,140.04,0.00),v40,fine,tPen\WObj:=wPaper;
    MoveL Offs(pOrigin,148.48,140.04,6.00),v60,z5,tPen\WObj:=wPaper;
    MoveL Offs(pOrigin,146.08,138.13,6.00),vTravel,z5,tPen\WObj:=wPaper;
    MoveL Offs(pOrigin,146.08,138.13,0.00),v60,z0,tPen\WObj:=wPaper;
    MoveL Offs(pOrigin,144.65,136.69,0.00),v40,z0,tPen\WObj:=wPaper;
    MoveL Offs(pOrigin,144.65,137.17,0.00),v40,z0,tPen\WObj:=wPaper;
    MoveL Offs(pOrigin,145.13,137.17,0.00),v40,z0,tPen\WObj:=wPaper;
    MoveL Offs(pOrigin,146.08,138.13,0.00),v40,z0,tPen\WObj:=wPaper;
    MoveL Offs(pOrigin,144.65,136.69,0.00),v40,z0,tPen\WObj:=wPaper;
    MoveL Offs(pOrigin,144.65,137.17,0.00),v40,z0,tPen\WObj:=wPaper;
    MoveL Offs(pOrigin,145.13,137.17,0.00),v40,z0,tPen\WObj:=wPaper;
    MoveL Offs(pOrigin,146.08,138.13,0.00),v40,fine,tPen\WObj:=wPaper;
    MoveL Offs(pOrigin,146.08,138.13,6.00),v60,z5,tPen\WObj:=wPaper;
    MoveL Offs(pOrigin,144.17,136.21,6.00),vTravel,z5,tPen\WObj:=wPaper;
    MoveL Offs(pOrigin,144.17,136.21,0.00),v60,z0,tPen\WObj:=wPaper;
    MoveL Offs(pOrigin,143.21,135.25,0.00),v40,z0,tPen\WObj:=wPaper;
    MoveL Offs(pOrigin,143.21,135.73,0.00),v40,z0,tPen\WObj:=wPaper;
    MoveL Offs(pOrigin,143.69,135.73,0.00),v40,z0,tPen\WObj:=wPaper;
    MoveL Offs(pOrigin,144.17,136.21,0.00),v40,z0,tPen\WObj:=wPaper;
    MoveL Offs(pOrigin,143.21,135.25,0.00),v40,z0,tPen\WObj:=wPaper;
    MoveL Offs(pOrigin,143.21,135.73,0.00),v40,z0,tPen\WObj:=wPaper;
    MoveL Offs(pOrigin,143.69,135.73,0.00),v40,z0,tPen\WObj:=wPaper;
    MoveL Offs(pOrigin,144.17,136.21,0.00),v40,fine,tPen\WObj:=wPaper;
    MoveL Offs(pOrigin,144.17,136.21,6.00),v60,z5,tPen\WObj:=wPaper;
    MoveL Offs(pOrigin,142.73,134.30,6.00),vTravel,z5,tPen\WObj:=wPaper;
    MoveL Offs(pOrigin,142.73,134.30,0.00),v60,z0,tPen\WObj:=wPaper;
    MoveL Offs(pOrigin,142.25,133.82,0.00),v40,z0,tPen\WObj:=wPaper;
    MoveL Offs(pOrigin,142.25,134.30,0.00),v40,z0,tPen\WObj:=wPaper;
    MoveL Offs(pOrigin,142.73,134.30,0.00),v40,z0,tPen\WObj:=wPaper;
    MoveL Offs(pOrigin,142.25,133.82,0.00),v40,z0,tPen\WObj:=wPaper;
    MoveL Offs(pOrigin,142.25,134.30,0.00),v40,z0,tPen\WObj:=wPaper;
    MoveL Offs(pOrigin,142.73,134.30,0.00),v40,fine,tPen\WObj:=wPaper;
    MoveL Offs(pOrigin,142.73,134.30,6.00),v60,z5,tPen\WObj:=wPaper;
    MoveL Offs(pOrigin,141.30,132.38,6.00),vTravel,z5,tPen\WObj:=wPaper;
    MoveL Offs(pOrigin,141.30,132.38,0.00),v60,z0,tPen\WObj:=wPaper;
    MoveL Offs(pOrigin,139.86,130.46,0.00),v40,z0,tPen\WObj:=wPaper;
    MoveL Offs(pOrigin,139.86,130.94,0.00),v40,z0,tPen\WObj:=wPaper;
    MoveL Offs(pOrigin,141.30,132.38,0.00),v40,z0,tPen\WObj:=wPaper;
    MoveL Offs(pOrigin,139.86,130.46,0.00),v40,z0,tPen\WObj:=wPaper;
    MoveL Offs(pOrigin,139.86,130.94,0.00),v40,z0,tPen\WObj:=wPaper;
    MoveL Offs(pOrigin,141.30,132.38,0.00),v40,fine,tPen\WObj:=wPaper;
    MoveL Offs(pOrigin,141.30,132.38,6.00),v60,z5,tPen\WObj:=wPaper;
    MoveL Offs(pOrigin,138.90,129.03,6.00),vTravel,z5,tPen\WObj:=wPaper;
    MoveL Offs(pOrigin,138.90,129.03,0.00),v60,z0,tPen\WObj:=wPaper;
    MoveL Offs(pOrigin,138.42,128.55,0.00),v40,z0,tPen\WObj:=wPaper;
    MoveL Offs(pOrigin,138.42,129.03,0.00),v40,z0,tPen\WObj:=wPaper;
    MoveL Offs(pOrigin,138.90,129.03,0.00),v40,z0,tPen\WObj:=wPaper;
    MoveL Offs(pOrigin,138.42,128.55,0.00),v40,z0,tPen\WObj:=wPaper;
    MoveL Offs(pOrigin,138.42,129.03,0.00),v40,z0,tPen\WObj:=wPaper;
  ENDPROC

  PROC DrawPart43()
    MoveL Offs(pOrigin,138.90,129.03,0.00),v40,fine,tPen\WObj:=wPaper;
    MoveL Offs(pOrigin,138.90,129.03,6.00),v60,z5,tPen\WObj:=wPaper;
    MoveL Offs(pOrigin,137.94,127.59,6.00),vTravel,z5,tPen\WObj:=wPaper;
    MoveL Offs(pOrigin,137.94,127.59,0.00),v60,z0,tPen\WObj:=wPaper;
    MoveL Offs(pOrigin,137.46,127.11,0.00),v40,z0,tPen\WObj:=wPaper;
    MoveL Offs(pOrigin,137.46,127.59,0.00),v40,z0,tPen\WObj:=wPaper;
    MoveL Offs(pOrigin,137.94,127.59,0.00),v40,z0,tPen\WObj:=wPaper;
    MoveL Offs(pOrigin,137.46,127.11,0.00),v40,z0,tPen\WObj:=wPaper;
    MoveL Offs(pOrigin,137.46,127.59,0.00),v40,z0,tPen\WObj:=wPaper;
    MoveL Offs(pOrigin,137.94,127.59,0.00),v40,fine,tPen\WObj:=wPaper;
    MoveL Offs(pOrigin,137.94,127.59,6.00),v60,z5,tPen\WObj:=wPaper;
    MoveL Offs(pOrigin,120.23,141.00,6.00),vTravel,z5,tPen\WObj:=wPaper;
    MoveL Offs(pOrigin,120.23,141.00,0.00),v60,z0,tPen\WObj:=wPaper;
    MoveL Offs(pOrigin,124.06,144.83,0.00),v40,z0,tPen\WObj:=wPaper;
    MoveL Offs(pOrigin,120.23,141.00,0.00),v40,fine,tPen\WObj:=wPaper;
    MoveL Offs(pOrigin,120.23,141.00,6.00),v60,z5,tPen\WObj:=wPaper;
    MoveL Offs(pOrigin,117.83,137.65,6.00),vTravel,z5,tPen\WObj:=wPaper;
    MoveL Offs(pOrigin,117.83,137.65,0.00),v60,z0,tPen\WObj:=wPaper;
    MoveL Offs(pOrigin,118.79,139.08,0.00),v40,z0,tPen\WObj:=wPaper;
    MoveL Offs(pOrigin,117.83,137.65,0.00),v40,z0,tPen\WObj:=wPaper;
    MoveL Offs(pOrigin,117.35,137.17,0.00),v40,z0,tPen\WObj:=wPaper;
    MoveL Offs(pOrigin,116.87,136.21,0.00),v40,z0,tPen\WObj:=wPaper;
    MoveL Offs(pOrigin,117.35,136.69,0.00),v40,z0,tPen\WObj:=wPaper;
    MoveL Offs(pOrigin,117.35,137.17,0.00),v40,z0,tPen\WObj:=wPaper;
    MoveL Offs(pOrigin,116.87,136.21,0.00),v40,z0,tPen\WObj:=wPaper;
    MoveL Offs(pOrigin,117.35,136.69,0.00),v40,z0,tPen\WObj:=wPaper;
    MoveL Offs(pOrigin,117.35,137.17,0.00),v40,fine,tPen\WObj:=wPaper;
    MoveL Offs(pOrigin,117.35,137.17,6.00),v60,z5,tPen\WObj:=wPaper;
    MoveL Offs(pOrigin,113.52,130.46,6.00),vTravel,z5,tPen\WObj:=wPaper;
    MoveL Offs(pOrigin,113.52,130.46,0.00),v60,z0,tPen\WObj:=wPaper;
    MoveL Offs(pOrigin,113.04,129.51,0.00),v40,z0,tPen\WObj:=wPaper;
    MoveL Offs(pOrigin,113.52,129.99,0.00),v40,z0,tPen\WObj:=wPaper;
    MoveL Offs(pOrigin,113.52,130.46,0.00),v40,z0,tPen\WObj:=wPaper;
    MoveL Offs(pOrigin,113.04,129.51,0.00),v40,z0,tPen\WObj:=wPaper;
    MoveL Offs(pOrigin,113.52,129.99,0.00),v40,z0,tPen\WObj:=wPaper;
    MoveL Offs(pOrigin,113.52,130.46,0.00),v40,fine,tPen\WObj:=wPaper;
    MoveL Offs(pOrigin,113.52,130.46,6.00),v60,z5,tPen\WObj:=wPaper;
    MoveL Offs(pOrigin,125.97,146.75,6.00),vTravel,z5,tPen\WObj:=wPaper;
    MoveL Offs(pOrigin,125.97,146.75,0.00),v60,z0,tPen\WObj:=wPaper;
    MoveL Offs(pOrigin,127.89,148.66,0.00),v40,z0,tPen\WObj:=wPaper;
    MoveL Offs(pOrigin,125.97,146.75,0.00),v40,fine,tPen\WObj:=wPaper;
    MoveL Offs(pOrigin,125.97,146.75,6.00),v60,z5,tPen\WObj:=wPaper;
    MoveL Offs(pOrigin,128.85,149.14,6.00),vTravel,z5,tPen\WObj:=wPaper;
    MoveL Offs(pOrigin,128.85,149.14,0.00),v60,z0,tPen\WObj:=wPaper;
    MoveL Offs(pOrigin,129.80,150.10,0.00),v40,z0,tPen\WObj:=wPaper;
    MoveL Offs(pOrigin,128.85,149.14,0.00),v40,fine,tPen\WObj:=wPaper;
    MoveL Offs(pOrigin,128.85,149.14,6.00),v60,z5,tPen\WObj:=wPaper;
    MoveL Offs(pOrigin,131.72,151.54,6.00),vTravel,z5,tPen\WObj:=wPaper;
    MoveL Offs(pOrigin,131.72,151.54,0.00),v60,z0,tPen\WObj:=wPaper;
    MoveL Offs(pOrigin,132.20,151.54,0.00),v40,z0,tPen\WObj:=wPaper;
    MoveL Offs(pOrigin,133.15,152.49,0.00),v40,z0,tPen\WObj:=wPaper;
    MoveL Offs(pOrigin,131.72,151.54,0.00),v40,z0,tPen\WObj:=wPaper;
    MoveL Offs(pOrigin,132.20,151.54,0.00),v40,z0,tPen\WObj:=wPaper;
    MoveL Offs(pOrigin,133.15,152.49,0.00),v40,z0,tPen\WObj:=wPaper;
    MoveL Offs(pOrigin,131.72,151.54,0.00),v40,fine,tPen\WObj:=wPaper;
    MoveL Offs(pOrigin,131.72,151.54,6.00),v60,z5,tPen\WObj:=wPaper;
    MoveL Offs(pOrigin,136.03,154.41,6.00),vTravel,z5,tPen\WObj:=wPaper;
    MoveL Offs(pOrigin,136.03,154.41,0.00),v60,z0,tPen\WObj:=wPaper;
    MoveL Offs(pOrigin,136.51,154.41,0.00),v40,z0,tPen\WObj:=wPaper;
    MoveL Offs(pOrigin,136.99,154.89,0.00),v40,z0,tPen\WObj:=wPaper;
    MoveL Offs(pOrigin,136.03,154.41,0.00),v40,z0,tPen\WObj:=wPaper;
    MoveL Offs(pOrigin,136.51,154.41,0.00),v40,z0,tPen\WObj:=wPaper;
    MoveL Offs(pOrigin,136.99,154.89,0.00),v40,z0,tPen\WObj:=wPaper;
    MoveL Offs(pOrigin,136.03,154.41,0.00),v40,fine,tPen\WObj:=wPaper;
    MoveL Offs(pOrigin,136.03,154.41,6.00),v60,z5,tPen\WObj:=wPaper;
    MoveL Offs(pOrigin,126.45,165.42,6.00),vTravel,z5,tPen\WObj:=wPaper;
    MoveL Offs(pOrigin,126.45,165.42,0.00),v60,z0,tPen\WObj:=wPaper;
    MoveL Offs(pOrigin,126.45,165.90,0.00),v40,z0,tPen\WObj:=wPaper;
    MoveL Offs(pOrigin,126.93,165.90,0.00),v40,z0,tPen\WObj:=wPaper;
    MoveL Offs(pOrigin,126.45,165.42,0.00),v40,z0,tPen\WObj:=wPaper;
    MoveL Offs(pOrigin,126.45,165.90,0.00),v40,z0,tPen\WObj:=wPaper;
    MoveL Offs(pOrigin,126.93,165.90,0.00),v40,z0,tPen\WObj:=wPaper;
    MoveL Offs(pOrigin,126.45,165.42,0.00),v40,fine,tPen\WObj:=wPaper;
    MoveL Offs(pOrigin,126.45,165.42,6.00),v60,z5,tPen\WObj:=wPaper;
    MoveL Offs(pOrigin,128.85,167.34,6.00),vTravel,z5,tPen\WObj:=wPaper;
    MoveL Offs(pOrigin,128.85,167.34,0.00),v60,z0,tPen\WObj:=wPaper;
    MoveL Offs(pOrigin,128.85,167.82,0.00),v40,z0,tPen\WObj:=wPaper;
    MoveL Offs(pOrigin,129.32,167.82,0.00),v40,z0,tPen\WObj:=wPaper;
    MoveL Offs(pOrigin,128.85,167.34,0.00),v40,z0,tPen\WObj:=wPaper;
    MoveL Offs(pOrigin,128.85,167.82,0.00),v40,z0,tPen\WObj:=wPaper;
    MoveL Offs(pOrigin,129.32,167.82,0.00),v40,z0,tPen\WObj:=wPaper;
    MoveL Offs(pOrigin,128.85,167.34,0.00),v40,fine,tPen\WObj:=wPaper;
    MoveL Offs(pOrigin,128.85,167.34,6.00),v60,z5,tPen\WObj:=wPaper;
    MoveL Offs(pOrigin,163.80,28.46,6.00),vTravel,z5,tPen\WObj:=wPaper;
    MoveL Offs(pOrigin,163.80,28.46,0.00),v60,z0,tPen\WObj:=wPaper;
    MoveL Offs(pOrigin,162.85,27.51,0.00),v40,z0,tPen\WObj:=wPaper;
    MoveL Offs(pOrigin,162.85,27.99,0.00),v40,z0,tPen\WObj:=wPaper;
    MoveL Offs(pOrigin,163.32,27.99,0.00),v40,z0,tPen\WObj:=wPaper;
    MoveL Offs(pOrigin,163.80,28.46,0.00),v40,z0,tPen\WObj:=wPaper;
    MoveL Offs(pOrigin,162.85,27.51,0.00),v40,z0,tPen\WObj:=wPaper;
    MoveL Offs(pOrigin,162.85,27.99,0.00),v40,z0,tPen\WObj:=wPaper;
    MoveL Offs(pOrigin,163.32,27.99,0.00),v40,z0,tPen\WObj:=wPaper;
    MoveL Offs(pOrigin,163.80,28.46,0.00),v40,fine,tPen\WObj:=wPaper;
    MoveL Offs(pOrigin,163.80,28.46,6.00),v60,z5,tPen\WObj:=wPaper;
    MoveL Offs(pOrigin,309.86,298.55,6.00),vTravel,z5,tPen\WObj:=wPaper;
    MoveL Offs(pOrigin,309.86,298.55,0.00),v60,z0,tPen\WObj:=wPaper;
    MoveL Offs(pOrigin,309.38,299.51,0.00),v40,z0,tPen\WObj:=wPaper;
    MoveL Offs(pOrigin,309.86,299.03,0.00),v40,z0,tPen\WObj:=wPaper;
    MoveL Offs(pOrigin,309.86,298.55,0.00),v40,z0,tPen\WObj:=wPaper;
    MoveL Offs(pOrigin,309.38,299.51,0.00),v40,z0,tPen\WObj:=wPaper;
    MoveL Offs(pOrigin,309.86,299.03,0.00),v40,z0,tPen\WObj:=wPaper;
    MoveL Offs(pOrigin,309.86,298.55,0.00),v40,fine,tPen\WObj:=wPaper;
    MoveL Offs(pOrigin,309.86,298.55,6.00),v60,z5,tPen\WObj:=wPaper;
    MoveL Offs(pOrigin,326.62,310.52,6.00),vTravel,z5,tPen\WObj:=wPaper;
    MoveL Offs(pOrigin,326.62,310.52,0.00),v60,z0,tPen\WObj:=wPaper;
    MoveL Offs(pOrigin,326.62,311.00,0.00),v40,z0,tPen\WObj:=wPaper;
    MoveL Offs(pOrigin,326.14,311.48,0.00),v40,z0,tPen\WObj:=wPaper;
    MoveL Offs(pOrigin,326.62,310.52,0.00),v40,z0,tPen\WObj:=wPaper;
    MoveL Offs(pOrigin,326.62,311.00,0.00),v40,z0,tPen\WObj:=wPaper;
    MoveL Offs(pOrigin,326.14,311.48,0.00),v40,z0,tPen\WObj:=wPaper;
    MoveL Offs(pOrigin,326.62,310.52,0.00),v40,fine,tPen\WObj:=wPaper;
    MoveL Offs(pOrigin,326.62,310.52,6.00),v60,z5,tPen\WObj:=wPaper;
  ENDPROC

ENDMODULE
